LIN {X 0,Y 448.468,Z 1012.095,A -85,B 0,C 180,E1 21481.185,E2 21481.185} C_VEL
LIN {X 0,Y 450.791,Z 994.348,A -85,B 0,C 180,E1 21478.882,E2 21478.882} C_VEL
LIN {X 0,Y 453.171,Z 976.212,A -85,B 0,C 180,E1 21476.826,E2 21476.826} C_VEL
LIN {X 0,Y 455.624,Z 956.598,A -85,B 0,C 180,E1 21474.938,E2 21474.938} C_VEL
LIN {X 0,Y 458.226,Z 934.729,A -85,B 0,C 180,E1 21473.126,E2 21473.126} C_VEL
LIN {X 0,Y 460.541,Z 914.08,A -85,B 0,C 180,E1 21471.667,E2 21471.667} C_VEL
LIN {X 0,Y 462.807,Z 891.263,A -85,B 0,C 180,E1 21470.327,E2 21470.327} C_VEL
LIN {X 0,Y 464.943,Z 868.015,A -85,B 0,C 180,E1 21469.198,E2 21469.198} C_VEL
LIN {X 0,Y 466.739,Z 845.323,A -85,B 0,C 180,E1 21468.323,E2 21468.323} C_VEL
LIN {X 0,Y 468.364,Z 820.403,A -85,B 0,C 180,E1 21467.596,E2 21467.596} C_VEL
LIN {X 0,Y 469.433,Z 794.902,A -85,B 0,C 180,E1 21467.062,E2 21467.062} C_VEL
LIN {X 0,Y 475.124,Z 590.761,A -85,B 0,C 180,E1 21463.377,E2 21463.377} C_VEL
LIN {X 0,Y 477.769,Z 494.434,A -85,B 0,C 180,E1 21461.609,E2 21461.609} C_VEL
LIN {X 0,Y 474.776,Z 465.725,A -85,B 0,C 180,E1 21460.637,E2 21460.637} C_VEL
LIN {X 0,Y 475.531,Z 455.632,A -85,B 0,C 180,E1 21460.006,E2 21460.006} C_VEL
LIN {X 0,Y 466.495,Z 437.235,A -85,B 0,C 180,E1 21457.496,E2 21457.496} C_VEL
LIN {X 0,Y 457.538,Z 420.696,A -85,B 0,C 180,E1 21454.928,E2 21454.928} C_VEL
LIN {X 0,Y 449.786,Z 407.184,A -85,B 0,C 180,E1 21452.544,E2 21452.544} C_VEL
LIN {X 0,Y 447.205,Z 402.648,A -85,B 0,C 180,E1 21451.695,E2 21451.695} C_VEL
LIN {X 0,Y 444.59,Z 398.544,A -85,B 0,C 180,E1 21450.847,E2 21450.847} C_VEL
LIN {X 0,Y 443.917,Z 397.22,A -85,B 0,C 180,E1 21450.599,E2 21450.599} C_VEL
LIN {X 0,Y 441.681,Z 394.126,A -85,B 0,C 180,E1 21449.885,E2 21449.885} C_VEL
LIN {X 0,Y 441.204,Z 392.302,A -85,B 0,C 180,E1 21449.514,E2 21449.514} C_VEL
LIN {X 0,Y 441.121,Z 392.05,A -85,B 0,C 180,E1 21445.941,E2 21445.941} C_VEL
LIN {X 0,Y 441.125,Z 392.099,A -85,B 0,C 180,E1 21442.242,E2 21442.242} C_VEL
LIN {X 0,Y 441.157,Z 392.047,A -85,B 0,C 180,E1 21438.636,E2 21438.636} C_VEL
LIN {X 0,Y 441.161,Z 392.066,A -85,B 0,C 180,E1 21434.973,E2 21434.973} C_VEL
LIN {X 0,Y 441.122,Z 392.06,A -85,B 0,C 180,E1 21431.373,E2 21431.373} C_VEL
LIN {X 0,Y 441.124,Z 392.081,A -85,B 0,C 180,E1 21427.554,E2 21427.554} C_VEL
LIN {X 0,Y 441.164,Z 392.078,A -85,B 0,C 180,E1 21424.028,E2 21424.028} C_VEL
LIN {X 0,Y 441.174,Z 392.079,A -85,B 0,C 180,E1 21420.259,E2 21420.259} C_VEL
LIN {X 0,Y 441.132,Z 392.084,A -85,B 0,C 180,E1 21416.621,E2 21416.621} C_VEL
LIN {X 0,Y 441.128,Z 392.084,A -85,B 0,C 180,E1 21412.969,E2 21412.969} C_VEL
LIN {X 0,Y 441.171,Z 392.08,A -85,B 0,C 180,E1 21409.421,E2 21409.421} C_VEL
LIN {X 0,Y 441.17,Z 392.083,A -85,B 0,C 180,E1 21405.697,E2 21405.697} C_VEL
LIN {X 0,Y 441.133,Z 392.089,A -85,B 0,C 180,E1 21402.046,E2 21402.046} C_VEL
LIN {X 0,Y 441.131,Z 392.086,A -85,B 0,C 180,E1 21398.318,E2 21398.318} C_VEL
LIN {X 0,Y 441.17,Z 392.081,A -85,B 0,C 180,E1 21394.728,E2 21394.728} C_VEL
LIN {X 0,Y 441.163,Z 392.055,A -85,B 0,C 180,E1 21391.135,E2 21391.135} C_VEL
LIN {X 0,Y 441.135,Z 392.085,A -85,B 0,C 180,E1 21387.476,E2 21387.476} C_VEL
LIN {X 0,Y 441.131,Z 392.048,A -85,B 0,C 180,E1 21383.731,E2 21383.731} C_VEL
LIN {X 0,Y 441.177,Z 392.355,A -85,B 0,C 180,E1 21381.087,E2 21381.087} C_VEL
LIN {X 0,Y 442.762,Z 395.916,A -85,B 0,C 180,E1 21380.276,E2 21380.276} C_VEL
LIN {X 0,Y 443.854,Z 397.437,A -85,B 0,C 180,E1 21379.889,E2 21379.889} C_VEL
LIN {X 0,Y 445.782,Z 401.239,A -85,B 0,C 180,E1 21379.085,E2 21379.085} C_VEL
LIN {X 0,Y 446.794,Z 403.101,A -85,B 0,C 180,E1 21378.687,E2 21378.687} C_VEL
LIN {X 0,Y 451.901,Z 412.956,A -85,B 0,C 180,E1 21376.694,E2 21376.694} C_VEL
LIN {X 0,Y 457.667,Z 424.557,A -85,B 0,C 180,E1 21374.531,E2 21374.531} C_VEL
LIN {X 0,Y 464.484,Z 439.37,A -85,B 0,C 180,E1 21372.026,E2 21372.026} C_VEL
LIN {X 0,Y 468.3,Z 448.451,A -85,B 0,C 180,E1 21370.633,E2 21370.633} C_VEL
LIN {X 0,Y 466.212,Z 469.982,A -85,B 0,C 180,E1 21368.876,E2 21368.876} C_VEL
LIN {X 0,Y 471.019,Z 499.481,A -85,B 0,C 180,E1 21367.741,E2 21367.741} C_VEL
LIN {X 0,Y 468.419,Z 640.813,A -85,B 0,C 180,E1 21365.511,E2 21365.511} C_VEL
LIN {X 0,Y 467.57,Z 648.523,A -85,B 0,C 180,E1 21365.47,E2 21365.47} C_VEL
LIN {X 0,Y 462.514,Z 669.112,A -85,B 0,C 180,E1 21365.661,E2 21365.661} C_VEL
LIN {X 0,Y 461.847,Z 675.731,A -85,B 0,C 180,E1 21365.619,E2 21365.619} C_VEL
LIN {X 0,Y 460.705,Z 743.485,A -85,B 0,C 180,E1 21364.531,E2 21364.531} C_VEL
LIN {X 0,Y 459.78,Z 763.748,A -85,B 0,C 180,E1 21363.979,E2 21363.979} C_VEL
LIN {X 0,Y 458.394,Z 783.122,A -85,B 0,C 180,E1 21363.232,E2 21363.232} C_VEL
LIN {X 0,Y 456.607,Z 801.726,A -85,B 0,C 180,E1 21362.297,E2 21362.297} C_VEL
LIN {X 0,Y 454.373,Z 820.148,A -85,B 0,C 180,E1 21361.129,E2 21361.129} C_VEL
LIN {X 0,Y 451.88,Z 837.225,A -85,B 0,C 180,E1 21359.785,E2 21359.785} C_VEL
LIN {X 0,Y 449.157,Z 853.741,A -85,B 0,C 180,E1 21358.22,E2 21358.22} C_VEL
LIN {X 0,Y 446.413,Z 869.137,A -85,B 0,C 180,E1 21356.469,E2 21356.469} C_VEL
LIN {X 0,Y 443.615,Z 883.656,A -85,B 0,C 180,E1 21354.502,E2 21354.502} C_VEL
LIN {X 0,Y 440.907,Z 897.352,A -85,B 0,C 180,E1 21352.254,E2 21352.254} C_VEL
LIN {X 0,Y 438.611,Z 908.804,A -85,B 0,C 180,E1 21349.995,E2 21349.995} C_VEL
LIN {X 0,Y 436.583,Z 919.459,A -85,B 0,C 180,E1 21347.459,E2 21347.459} C_VEL
LIN {X 0,Y 434.978,Z 928.589,A -85,B 0,C 180,E1 21344.783,E2 21344.783} C_VEL
LIN {X 0,Y 433.854,Z 935.893,A -85,B 0,C 180,E1 21342.106,E2 21342.106} C_VEL
LIN {X 0,Y 433.096,Z 942.058,A -85,B 0,C 180,E1 21339.166,E2 21339.166} C_VEL
LIN {X 0,Y 432.688,Z 946.439,A -85,B 0,C 180,E1 21336.235,E2 21336.235} C_VEL
LIN {X 0,Y 432.469,Z 949.098,A -85,B 0,C 180,E1 21333.314,E2 21333.314} C_VEL
LIN {X 0,Y 432.408,Z 950.106,A -85,B 0,C 180,E1 21330.53,E2 21330.53} C_VEL
LIN {X 0,Y 432.438,Z 949.614,A -85,B 0,C 180,E1 21327.615,E2 21327.615} C_VEL
LIN {X 0,Y 432.577,Z 947.513,A -85,B 0,C 180,E1 21324.695,E2 21324.695} C_VEL
LIN {X 0,Y 432.899,Z 943.973,A -85,B 0,C 180,E1 21321.901,E2 21321.901} C_VEL
LIN {X 0,Y 433.461,Z 938.858,A -85,B 0,C 180,E1 21319.097,E2 21319.097} C_VEL
LIN {X 0,Y 434.522,Z 931.627,A -85,B 0,C 180,E1 21316.154,E2 21316.154} C_VEL
LIN {X 0,Y 435.898,Z 923.218,A -85,B 0,C 180,E1 21313.475,E2 21313.475} C_VEL
LIN {X 0,Y 437.744,Z 913.352,A -85,B 0,C 180,E1 21310.936,E2 21310.936} C_VEL
LIN {X 0,Y 439.944,Z 902.052,A -85,B 0,C 180,E1 21308.537,E2 21308.537} C_VEL
LIN {X 0,Y 442.345,Z 890.111,A -85,B 0,C 180,E1 21306.416,E2 21306.416} C_VEL
LIN {X 0,Y 445.131,Z 875.915,A -85,B 0,C 180,E1 21304.309,E2 21304.309} C_VEL
LIN {X 0,Y 448.018,Z 860.412,A -85,B 0,C 180,E1 21302.406,E2 21302.406} C_VEL
LIN {X 0,Y 450.706,Z 844.615,A -85,B 0,C 180,E1 21300.787,E2 21300.787} C_VEL
LIN {X 0,Y 453.397,Z 827.134,A -85,B 0,C 180,E1 21299.301,E2 21299.301} C_VEL
LIN {X 0,Y 455.721,Z 809.616,A -85,B 0,C 180,E1 21298.078,E2 21298.078} C_VEL
LIN {X 0,Y 457.698,Z 791.119,A -85,B 0,C 180,E1 21297.047,E2 21297.047} C_VEL
LIN {X 0,Y 459.274,Z 772.031,A -85,B 0,C 180,E1 21296.223,E2 21296.223} C_VEL
LIN {X 0,Y 460.396,Z 751.626,A -85,B 0,C 180,E1 21295.574,E2 21295.574} C_VEL
LIN {X 0,Y 460.968,Z 731.073,A -85,B 0,C 180,E1 21295.147,E2 21295.147} C_VEL
LIN {X 0,Y 465.125,Z 504.024,A -85,B 0,C 180,E1 21291.563,E2 21291.563} C_VEL
LIN {X 0,Y 465.006,Z 498.899,A -85,B 0,C 180,E1 21291.45,E2 21291.45} C_VEL
LIN {X 0,Y 460.181,Z 468.723,A -85,B 0,C 180,E1 21290.217,E2 21290.217} C_VEL
LIN {X 0,Y 461.91,Z 451.947,A -85,B 0,C 180,E1 21288.792,E2 21288.792} C_VEL
LIN {X 0,Y 454.83,Z 435.65,A -85,B 0,C 180,E1 21286.141,E2 21286.141} C_VEL
LIN {X 0,Y 447.451,Z 420.273,A -85,B 0,C 180,E1 21283.316,E2 21283.316} C_VEL
LIN {X 0,Y 440.681,Z 407.247,A -85,B 0,C 180,E1 21280.63,E2 21280.63} C_VEL
LIN {X 0,Y 437.714,Z 401.938,A -85,B 0,C 180,E1 21279.423,E2 21279.423} C_VEL
LIN {X 0,Y 435.539,Z 397.815,A -85,B 0,C 180,E1 21278.472,E2 21278.472} C_VEL
LIN {X 0,Y 433.601,Z 394.615,A -85,B 0,C 180,E1 21277.668,E2 21277.668} C_VEL
LIN {X 0,Y 433.24,Z 393.102,A -85,B 0,C 180,E1 21277.234,E2 21277.234} C_VEL
LIN {X 0,Y 433.25,Z 393.077,A -85,B 0,C 180,E1 21273.475,E2 21273.475} C_VEL
LIN {X 0,Y 433.203,Z 393.029,A -85,B 0,C 180,E1 21269.751,E2 21269.751} C_VEL
LIN {X 0,Y 433.199,Z 393.076,A -85,B 0,C 180,E1 21266.011,E2 21266.011} C_VEL
LIN {X 0,Y 433.206,Z 393.071,A -85,B 0,C 180,E1 21262.242,E2 21262.242} C_VEL
LIN {X 0,Y 433.243,Z 393.068,A -85,B 0,C 180,E1 21258.572,E2 21258.572} C_VEL
LIN {X 0,Y 433.227,Z 393.068,A -85,B 0,C 180,E1 21254.844,E2 21254.844} C_VEL
LIN {X 0,Y 433.195,Z 393.07,A -85,B 0,C 180,E1 21251.18,E2 21251.18} C_VEL
LIN {X 0,Y 433.193,Z 393.071,A -85,B 0,C 180,E1 21247.427,E2 21247.427} C_VEL
LIN {X 0,Y 433.23,Z 393.068,A -85,B 0,C 180,E1 21243.838,E2 21243.838} C_VEL
LIN {X 0,Y 433.248,Z 393.067,A -85,B 0,C 180,E1 21240,E2 21240} C_VEL
LIN {X 0,Y 433.203,Z 393.073,A -85,B 0,C 180,E1 21236.295,E2 21236.295} C_VEL
LIN {X 0,Y 433.187,Z 393.073,A -85,B 0,C 180,E1 21232.574,E2 21232.574} C_VEL
LIN {X 0,Y 433.195,Z 393.053,A -85,B 0,C 180,E1 21228.821,E2 21228.821} C_VEL
LIN {X 0,Y 433.239,Z 393.044,A -85,B 0,C 180,E1 21225.157,E2 21225.157} C_VEL
LIN {X 0,Y 433.213,Z 393.034,A -85,B 0,C 180,E1 21221.428,E2 21221.428} C_VEL
LIN {X 0,Y 433.188,Z 393.084,A -85,B 0,C 180,E1 21217.755,E2 21217.755} C_VEL
LIN {X 0,Y 433.18,Z 393.037,A -85,B 0,C 180,E1 21213.882,E2 21213.882} C_VEL
LIN {X 0,Y 433.206,Z 393.185,A -85,B 0,C 180,E1 21212.061,E2 21212.061} C_VEL
LIN {X 0,Y 433.375,Z 394.077,A -85,B 0,C 180,E1 21211.774,E2 21211.774} C_VEL
LIN {X 0,Y 434.939,Z 397.128,A -85,B 0,C 180,E1 21211.135,E2 21211.135} C_VEL
LIN {X 0,Y 436.493,Z 398.918,A -85,B 0,C 180,E1 21210.647,E2 21210.647} C_VEL
LIN {X 0,Y 438.48,Z 402.68,A -85,B 0,C 180,E1 21209.891,E2 21209.891} C_VEL
LIN {X 0,Y 439.64,Z 404.191,A -85,B 0,C 180,E1 21209.526,E2 21209.526} C_VEL
LIN {X 0,Y 448.134,Z 418.764,A -85,B 0,C 180,E1 21206.711,E2 21206.711} C_VEL
LIN {X 0,Y 457.182,Z 435.066,A -85,B 0,C 180,E1 21203.964,E2 21203.964} C_VEL
LIN {X 0,Y 466.517,Z 453.526,A -85,B 0,C 180,E1 21201.258,E2 21201.258} C_VEL
LIN {X 0,Y 469.372,Z 459.759,A -85,B 0,C 180,E1 21200.437,E2 21200.437} C_VEL
LIN {X 0,Y 468.908,Z 467.207,A -85,B 0,C 180,E1 21200.003,E2 21200.003} C_VEL
LIN {X 0,Y 471.972,Z 498.397,A -85,B 0,C 180,E1 21198.963,E2 21198.963} C_VEL
LIN {X 0,Y 465.873,Z 694.074,A -85,B 0,C 180,E1 21195.358,E2 21195.358} C_VEL
LIN {X 0,Y 462.333,Z 810.411,A -85,B 0,C 180,E1 21193.203,E2 21193.203} C_VEL
LIN {X 0,Y 460.677,Z 834.598,A -85,B 0,C 180,E1 21192.553,E2 21192.553} C_VEL
LIN {X 0,Y 458.633,Z 859.758,A -85,B 0,C 180,E1 21191.63,E2 21191.63} C_VEL
LIN {X 0,Y 456.391,Z 883.845,A -85,B 0,C 180,E1 21190.518,E2 21190.518} C_VEL
LIN {X 0,Y 454.058,Z 905.996,A -85,B 0,C 180,E1 21189.258,E2 21189.258} C_VEL
LIN {X 0,Y 451.451,Z 929.158,A -85,B 0,C 180,E1 21187.682,E2 21187.682} C_VEL
LIN {X 0,Y 448.984,Z 949.425,A -85,B 0,C 180,E1 21186.063,E2 21186.063} C_VEL
LIN {X 0,Y 446.433,Z 969.107,A -85,B 0,C 180,E1 21184.205,E2 21184.205} C_VEL
LIN {X 0,Y 443.953,Z 987.875,A -85,B 0,C 180,E1 21182.177,E2 21182.177} C_VEL
LIN {X 0,Y 441.759,Z 1003.879,A -85,B 0,C 180,E1 21180.164,E2 21180.164} C_VEL
LIN {X 0,Y 439.529,Z 1020.382,A -85,B 0,C 180,E1 21177.797,E2 21177.797} C_VEL
LIN {X 0,Y 437.627,Z 1034.57,A -85,B 0,C 180,E1 21175.438,E2 21175.438} C_VEL
LIN {X 0,Y 436.501,Z 1043.063,A -85,B 0,C 180,E1 21173.775,E2 21173.775} C_VEL
LIN {X 0,Y 434.82,Z 1055.286,A -85,B 0,C 180,E1 21170.881,E2 21170.881} C_VEL
LIN {X 0,Y 433.661,Z 1065.058,A -85,B 0,C 180,E1 21168.135,E2 21168.135} C_VEL
LIN {X 0,Y 432.778,Z 1074.344,A -85,B 0,C 180,E1 21164.996,E2 21164.996} C_VEL
LIN {X 0,Y 432.319,Z 1080.863,A -85,B 0,C 180,E1 21162.285,E2 21162.285} C_VEL
LIN {X 0,Y 432.046,Z 1086.635,A -85,B 0,C 180,E1 21159.189,E2 21159.189} C_VEL
LIN {X 0,Y 431.946,Z 1090.278,A -85,B 0,C 180,E1 21156.513,E2 21156.513} C_VEL
LIN {X 0,Y 431.89,Z 1092.916,A -85,B 0,C 180,E1 21153.451,E2 21153.451} C_VEL
LIN {X 0,Y 431.89,Z 1093.849,A -85,B 0,C 180,E1 21150.929,E2 21150.929} C_VEL
LIN {X 0,Y 431.906,Z 1093.69,A -85,B 0,C 180,E1 21148.143,E2 21148.143} C_VEL
LIN {X 0,Y 431.911,Z 1091.954,A -85,B 0,C 180,E1 21145.219,E2 21145.219} C_VEL
LIN {X 0,Y 431.947,Z 1089.16,A -85,B 0,C 180,E1 21142.552,E2 21142.552} C_VEL
LIN {X 0,Y 432.131,Z 1084.335,A -85,B 0,C 180,E1 21139.468,E2 21139.468} C_VEL
LIN {X 0,Y 432.457,Z 1078.689,A -85,B 0,C 180,E1 21136.745,E2 21136.745} C_VEL
LIN {X 0,Y 433.109,Z 1070.549,A -85,B 0,C 180,E1 21133.641,E2 21133.641} C_VEL
LIN {X 0,Y 434.063,Z 1061.522,A -85,B 0,C 180,E1 21130.808,E2 21130.808} C_VEL
LIN {X 0,Y 435.397,Z 1050.859,A -85,B 0,C 180,E1 21128.018,E2 21128.018} C_VEL
LIN {X 0,Y 436.867,Z 1040.444,A -85,B 0,C 180,E1 21125.671,E2 21125.671} C_VEL
LIN {X 0,Y 438.484,Z 1028.182,A -85,B 0,C 180,E1 21123.453,E2 21123.453} C_VEL
LIN {X 0,Y 440.51,Z 1012.885,A -85,B 0,C 180,E1 21121.088,E2 21121.088} C_VEL
LIN {X 0,Y 442.927,Z 995.3,A -85,B 0,C 180,E1 21118.721,E2 21118.721} C_VEL
LIN {X 0,Y 445.296,Z 977.664,A -85,B 0,C 180,E1 21116.681,E2 21116.681} C_VEL
LIN {X 0,Y 447.942,Z 957.612,A -85,B 0,C 180,E1 21114.681,E2 21114.681} C_VEL
LIN {X 0,Y 450.477,Z 937.455,A -85,B 0,C 180,E1 21112.943,E2 21112.943} C_VEL
LIN {X 0,Y 452.963,Z 916.014,A -85,B 0,C 180,E1 21111.389,E2 21111.389} C_VEL
LIN {X 0,Y 455.519,Z 892.134,A -85,B 0,C 180,E1 21109.929,E2 21109.929} C_VEL
LIN {X 0,Y 457.861,Z 868.453,A -85,B 0,C 180,E1 21108.738,E2 21108.738} C_VEL
LIN {X 0,Y 459.897,Z 845.034,A -85,B 0,C 180,E1 21107.8,E2 21107.8} C_VEL
LIN {X 0,Y 461.703,Z 820.565,A -85,B 0,C 180,E1 21107.048,E2 21107.048} C_VEL
LIN {X 0,Y 462.89,Z 796.443,A -85,B 0,C 180,E1 21106.513,E2 21106.513} C_VEL
LIN {X 0,Y 469.226,Z 586.155,A -85,B 0,C 180,E1 21102.65,E2 21102.65} C_VEL
LIN {X 0,Y 471.857,Z 495.824,A -85,B 0,C 180,E1 21100.973,E2 21100.973} C_VEL
LIN {X 0,Y 468.83,Z 465.707,A -85,B 0,C 180,E1 21099.935,E2 21099.935} C_VEL
LIN {X 0,Y 469.264,Z 459.399,A -85,B 0,C 180,E1 21099.528,E2 21099.528} C_VEL
LIN {X 0,Y 460.765,Z 442.036,A -85,B 0,C 180,E1 21097.103,E2 21097.103} C_VEL
LIN {X 0,Y 451.956,Z 425.626,A -85,B 0,C 180,E1 21094.495,E2 21094.495} C_VEL
LIN {X 0,Y 444.665,Z 412.9,A -85,B 0,C 180,E1 21092.202,E2 21092.202} C_VEL
LIN {X 0,Y 441.33,Z 407.353,A -85,B 0,C 180,E1 21091.1,E2 21091.1} C_VEL
LIN {X 0,Y 439.258,Z 403.53,A -85,B 0,C 180,E1 21090.352,E2 21090.352} C_VEL
LIN {X 0,Y 437.001,Z 400.277,A -85,B 0,C 180,E1 21089.605,E2 21089.605} C_VEL
LIN {X 0,Y 436.11,Z 398.272,A -85,B 0,C 180,E1 21089.231,E2 21089.231} C_VEL
LIN {X 0,Y 433.852,Z 395.425,A -85,B 0,C 180,E1 21088.493,E2 21088.493} C_VEL
LIN {X 0,Y 433.221,Z 393.312,A -85,B 0,C 180,E1 21088.049,E2 21088.049} C_VEL
LIN {X 0,Y 433.199,Z 393.038,A -85,B 0,C 180,E1 21084.693,E2 21084.693} C_VEL
LIN {X 0,Y 433.235,Z 393.042,A -85,B 0,C 180,E1 21081.102,E2 21081.102} C_VEL
LIN {X 0,Y 433.202,Z 393.07,A -85,B 0,C 180,E1 21077.321,E2 21077.321} C_VEL
LIN {X 0,Y 433.178,Z 393.028,A -85,B 0,C 180,E1 21073.649,E2 21073.649} C_VEL
LIN {X 0,Y 433.2,Z 393.081,A -85,B 0,C 180,E1 21069.968,E2 21069.968} C_VEL
LIN {X 0,Y 433.247,Z 393.074,A -85,B 0,C 180,E1 21066.36,E2 21066.36} C_VEL
LIN {X 0,Y 433.219,Z 393.081,A -85,B 0,C 180,E1 21062.513,E2 21062.513} C_VEL
LIN {X 0,Y 433.188,Z 393.085,A -85,B 0,C 180,E1 21058.942,E2 21058.942} C_VEL
LIN {X 0,Y 433.192,Z 393.086,A -85,B 0,C 180,E1 21055.101,E2 21055.101} C_VEL
LIN {X 0,Y 433.233,Z 393.076,A -85,B 0,C 180,E1 21051.506,E2 21051.506} C_VEL
LIN {X 0,Y 433.233,Z 393.074,A -85,B 0,C 180,E1 21047.741,E2 21047.741} C_VEL
LIN {X 0,Y 433.192,Z 393.079,A -85,B 0,C 180,E1 21044.195,E2 21044.195} C_VEL
LIN {X 0,Y 433.192,Z 393.083,A -85,B 0,C 180,E1 21040.343,E2 21040.343} C_VEL
LIN {X 0,Y 433.222,Z 393.081,A -85,B 0,C 180,E1 21036.719,E2 21036.719} C_VEL
LIN {X 0,Y 433.25,Z 393.083,A -85,B 0,C 180,E1 21032.958,E2 21032.958} C_VEL
LIN {X 0,Y 433.198,Z 393.03,A -85,B 0,C 180,E1 21029.33,E2 21029.33} C_VEL
LIN {X 0,Y 433.193,Z 393.059,A -85,B 0,C 180,E1 21025.722,E2 21025.722} C_VEL
LIN {X 0,Y 433.275,Z 393.272,A -85,B 0,C 180,E1 21022.547,E2 21022.547} C_VEL
LIN {X 0,Y 434.562,Z 396.641,A -85,B 0,C 180,E1 21021.762,E2 21021.762} C_VEL
LIN {X 0,Y 436.025,Z 398.504,A -85,B 0,C 180,E1 21021.23,E2 21021.23} C_VEL
LIN {X 0,Y 437.837,Z 402.121,A -85,B 0,C 180,E1 21020.421,E2 21020.421} C_VEL
LIN {X 0,Y 439.101,Z 404.577,A -85,B 0,C 180,E1 21019.878,E2 21019.878} C_VEL
LIN {X 0,Y 441.467,Z 408.736,A -85,B 0,C 180,E1 21018.943,E2 21018.943} C_VEL
LIN {X 0,Y 447.932,Z 421.252,A -85,B 0,C 180,E1 21016.39,E2 21016.39} C_VEL
LIN {X 0,Y 455.311,Z 436.855,A -85,B 0,C 180,E1 21013.558,E2 21013.558} C_VEL
LIN {X 0,Y 461.991,Z 452.277,A -85,B 0,C 180,E1 21011.069,E2 21011.069} C_VEL
LIN {X 0,Y 460.191,Z 469.857,A -85,B 0,C 180,E1 21009.622,E2 21009.622} C_VEL
LIN {X 0,Y 465.187,Z 501.003,A -85,B 0,C 180,E1 21008.394,E2 21008.394} C_VEL
LIN {X 0,Y 461.847,Z 675.731,A -85,B 0,C 180,E1 21005.619,E2 21005.619} C_VEL
LIN {X 0,Y 460.984,Z 683.439,A -85,B 0,C 180,E1 21005.58,E2 21005.58} C_VEL
LIN {X 0,Y 455.916,Z 704.017,A -85,B 0,C 180,E1 21005.776,E2 21005.776} C_VEL
LIN {X 0,Y 455.217,Z 710.635,A -85,B 0,C 180,E1 21005.736,E2 21005.736} C_VEL
LIN {X 0,Y 454.534,Z 745.79,A -85,B 0,C 180,E1 21005.136,E2 21005.136} C_VEL
LIN {X 0,Y 453.54,Z 766.188,A -85,B 0,C 180,E1 21004.56,E2 21004.56} C_VEL
LIN {X 0,Y 452.058,Z 785.284,A -85,B 0,C 180,E1 21003.798,E2 21003.798} C_VEL
LIN {X 0,Y 450.103,Z 804.155,A -85,B 0,C 180,E1 21002.822,E2 21002.822} C_VEL
LIN {X 0,Y 447.8,Z 822.219,A -85,B 0,C 180,E1 21001.649,E2 21001.649} C_VEL
LIN {X 0,Y 445.18,Z 839.286,A -85,B 0,C 180,E1 21000.28,E2 21000.28} C_VEL
LIN {X 0,Y 442.37,Z 855.414,A -85,B 0,C 180,E1 20998.72,E2 20998.72} C_VEL
LIN {X 0,Y 439.448,Z 870.944,A -85,B 0,C 180,E1 20996.922,E2 20996.922} C_VEL
LIN {X 0,Y 436.702,Z 884.518,A -85,B 0,C 180,E1 20995.06,E2 20995.06} C_VEL
LIN {X 0,Y 433.977,Z 897.535,A -85,B 0,C 180,E1 20992.915,E2 20992.915} C_VEL
LIN {X 0,Y 431.439,Z 909.484,A -85,B 0,C 180,E1 20990.565,E2 20990.565} C_VEL
LIN {X 0,Y 429.187,Z 920.585,A -85,B 0,C 180,E1 20987.91,E2 20987.91} C_VEL
LIN {X 0,Y 427.435,Z 929.8,A -85,B 0,C 180,E1 20985.188,E2 20985.188} C_VEL
LIN {X 0,Y 426.209,Z 937.166,A -85,B 0,C 180,E1 20982.464,E2 20982.464} C_VEL
LIN {X 0,Y 425.364,Z 943.114,A -85,B 0,C 180,E1 20979.607,E2 20979.607} C_VEL
LIN {X 0,Y 424.878,Z 947.533,A -85,B 0,C 180,E1 20976.622,E2 20976.622} C_VEL
LIN {X 0,Y 424.62,Z 950.195,A -85,B 0,C 180,E1 20973.78,E2 20973.78} C_VEL
LIN {X 0,Y 424.534,Z 951.432,A -85,B 0,C 180,E1 20970.81,E2 20970.81} C_VEL
LIN {X 0,Y 424.558,Z 951.106,A -85,B 0,C 180,E1 20967.841,E2 20967.841} C_VEL
LIN {X 0,Y 424.706,Z 949.346,A -85,B 0,C 180,E1 20965.003,E2 20965.003} C_VEL
LIN {X 0,Y 425.049,Z 945.883,A -85,B 0,C 180,E1 20962.022,E2 20962.022} C_VEL
LIN {X 0,Y 425.668,Z 940.742,A -85,B 0,C 180,E1 20959.068,E2 20959.068} C_VEL
LIN {X 0,Y 426.675,Z 934.284,A -85,B 0,C 180,E1 20956.309,E2 20956.309} C_VEL
LIN {X 0,Y 428.088,Z 926.192,A -85,B 0,C 180,E1 20953.584,E2 20953.584} C_VEL
LIN {X 0,Y 429.983,Z 916.692,A -85,B 0,C 180,E1 20951.001,E2 20951.001} C_VEL
LIN {X 0,Y 432.235,Z 905.82,A -85,B 0,C 180,E1 20948.562,E2 20948.562} C_VEL
LIN {X 0,Y 434.946,Z 892.994,A -85,B 0,C 180,E1 20946.196,E2 20946.196} C_VEL
LIN {X 0,Y 437.714,Z 879.534,A -85,B 0,C 180,E1 20944.132,E2 20944.132} C_VEL
LIN {X 0,Y 440.615,Z 864.947,A -85,B 0,C 180,E1 20942.252,E2 20942.252} C_VEL
LIN {X 0,Y 443.487,Z 849.341,A -85,B 0,C 180,E1 20940.561,E2 20940.561} C_VEL
LIN {X 0,Y 446.277,Z 832.59,A -85,B 0,C 180,E1 20939.057,E2 20939.057} C_VEL
LIN {X 0,Y 448.798,Z 814.844,A -85,B 0,C 180,E1 20937.753,E2 20937.753} C_VEL
LIN {X 0,Y 450.993,Z 796.221,A -85,B 0,C 180,E1 20936.645,E2 20936.645} C_VEL
LIN {X 0,Y 452.798,Z 776.87,A -85,B 0,C 180,E1 20935.745,E2 20935.745} C_VEL
LIN {X 0,Y 454.099,Z 757.056,A -85,B 0,C 180,E1 20935.062,E2 20935.062} C_VEL
LIN {X 0,Y 454.763,Z 736.951,A -85,B 0,C 180,E1 20934.596,E2 20934.596} C_VEL
LIN {X 0,Y 459.428,Z 501.652,A -85,B 0,C 180,E1 20930.825,E2 20930.825} C_VEL
LIN {X 0,Y 454.252,Z 468.861,A -85,B 0,C 180,E1 20929.467,E2 20929.467} C_VEL
LIN {X 0,Y 455.628,Z 455.879,A -85,B 0,C 180,E1 20928.35,E2 20928.35} C_VEL
LIN {X 0,Y 448.298,Z 438.984,A -85,B 0,C 180,E1 20925.538,E2 20925.538} C_VEL
LIN {X 0,Y 441.704,Z 425.283,A -85,B 0,C 180,E1 20922.95,E2 20922.95} C_VEL
LIN {X 0,Y 435.753,Z 413.46,A -85,B 0,C 180,E1 20920.494,E2 20920.494} C_VEL
LIN {X 0,Y 432.121,Z 407.113,A -85,B 0,C 180,E1 20919.004,E2 20919.004} C_VEL
LIN {X 0,Y 430.277,Z 403.623,A -85,B 0,C 180,E1 20918.179,E2 20918.179} C_VEL
LIN {X 0,Y 428.446,Z 400.267,A -85,B 0,C 180,E1 20917.356,E2 20917.356} C_VEL
LIN {X 0,Y 427.9,Z 399.033,A -85,B 0,C 180,E1 20917.075,E2 20917.075} C_VEL
LIN {X 0,Y 425.896,Z 396.306,A -85,B 0,C 180,E1 20916.272,E2 20916.272} C_VEL
LIN {X 0,Y 425.331,Z 394.346,A -85,B 0,C 180,E1 20915.804,E2 20915.804} C_VEL
LIN {X 0,Y 425.258,Z 394.04,A -85,B 0,C 180,E1 20914.353,E2 20914.353} C_VEL
LIN {X 0,Y 425.265,Z 394.016,A -85,B 0,C 180,E1 20910.624,E2 20910.624} C_VEL
LIN {X 0,Y 425.311,Z 394.072,A -85,B 0,C 180,E1 20906.983,E2 20906.983} C_VEL
LIN {X 0,Y 425.302,Z 394.065,A -85,B 0,C 180,E1 20903.117,E2 20903.117} C_VEL
LIN {X 0,Y 425.269,Z 394.066,A -85,B 0,C 180,E1 20899.361,E2 20899.361} C_VEL
LIN {X 0,Y 425.257,Z 394.066,A -85,B 0,C 180,E1 20895.688,E2 20895.688} C_VEL
LIN {X 0,Y 425.281,Z 394.061,A -85,B 0,C 180,E1 20892.028,E2 20892.028} C_VEL
LIN {X 0,Y 425.313,Z 394.058,A -85,B 0,C 180,E1 20888.219,E2 20888.219} C_VEL
LIN {X 0,Y 425.28,Z 394.064,A -85,B 0,C 180,E1 20884.45,E2 20884.45} C_VEL
LIN {X 0,Y 425.253,Z 394.071,A -85,B 0,C 180,E1 20880.809,E2 20880.809} C_VEL
LIN {X 0,Y 425.252,Z 394.069,A -85,B 0,C 180,E1 20876.9,E2 20876.9} C_VEL
LIN {X 0,Y 425.279,Z 394.065,A -85,B 0,C 180,E1 20873.25,E2 20873.25} C_VEL
LIN {X 0,Y 425.297,Z 394.058,A -85,B 0,C 180,E1 20869.571,E2 20869.571} C_VEL
LIN {X 0,Y 425.257,Z 394.019,A -85,B 0,C 180,E1 20865.847,E2 20865.847} C_VEL
LIN {X 0,Y 425.246,Z 394.041,A -85,B 0,C 180,E1 20862.202,E2 20862.202} C_VEL
LIN {X 0,Y 425.263,Z 394.042,A -85,B 0,C 180,E1 20858.483,E2 20858.483} C_VEL
LIN {X 0,Y 425.294,Z 394.015,A -85,B 0,C 180,E1 20854.816,E2 20854.816} C_VEL
LIN {X 0,Y 425.294,Z 394.362,A -85,B 0,C 180,E1 20853.545,E2 20853.545} C_VEL
LIN {X 0,Y 426.96,Z 398.008,A -85,B 0,C 180,E1 20852.678,E2 20852.678} C_VEL
LIN {X 0,Y 428.482,Z 399.64,A -85,B 0,C 180,E1 20852.178,E2 20852.178} C_VEL
LIN {X 0,Y 430.326,Z 403.372,A -85,B 0,C 180,E1 20851.404,E2 20851.404} C_VEL
LIN {X 0,Y 431.832,Z 405.265,A -85,B 0,C 180,E1 20850.907,E2 20850.907} C_VEL
LIN {X 0,Y 434.233,Z 409.398,A -85,B 0,C 180,E1 20850.023,E2 20850.023} C_VEL
LIN {X 0,Y 438.552,Z 416.859,A -85,B 0,C 180,E1 20848.506,E2 20848.506} C_VEL
LIN {X 0,Y 443.384,Z 425.066,A -85,B 0,C 180,E1 20846.926,E2 20846.926} C_VEL
LIN {X 0,Y 451.941,Z 440.635,A -85,B 0,C 180,E1 20844.264,E2 20844.264} C_VEL
LIN {X 0,Y 461.147,Z 459.091,A -85,B 0,C 180,E1 20841.518,E2 20841.518} C_VEL
LIN {X 0,Y 463.174,Z 463.478,A -85,B 0,C 180,E1 20840.925,E2 20840.925} C_VEL
LIN {X 0,Y 463.074,Z 467.74,A -85,B 0,C 180,E1 20840.701,E2 20840.701} C_VEL
LIN {X 0,Y 466.123,Z 499.761,A -85,B 0,C 180,E1 20839.614,E2 20839.614} C_VEL
LIN {X 0,Y 459.725,Z 693.452,A -85,B 0,C 180,E1 20836.004,E2 20836.004} C_VEL
LIN {X 0,Y 455.951,Z 809.256,A -85,B 0,C 180,E1 20833.823,E2 20833.823} C_VEL
LIN {X 0,Y 454.215,Z 833.206,A -85,B 0,C 180,E1 20833.172,E2 20833.172} C_VEL
LIN {X 0,Y 452.033,Z 857.97,A -85,B 0,C 180,E1 20832.255,E2 20832.255} C_VEL
LIN {X 0,Y 449.685,Z 881.129,A -85,B 0,C 180,E1 20831.159,E2 20831.159} C_VEL
LIN {X 0,Y 446.945,Z 904.721,A -85,B 0,C 180,E1 20829.778,E2 20829.778} C_VEL
LIN {X 0,Y 444.165,Z 928.038,A -85,B 0,C 180,E1 20828.165,E2 20828.165} C_VEL
LIN {X 0,Y 441.538,Z 948.91,A -85,B 0,C 180,E1 20826.472,E2 20826.472} C_VEL
LIN {X 0,Y 438.845,Z 968.868,A -85,B 0,C 180,E1 20824.564,E2 20824.564} C_VEL
LIN {X 0,Y 436.154,Z 988.289,A -85,B 0,C 180,E1 20822.402,E2 20822.402} C_VEL
LIN {X 0,Y 433.859,Z 1004.571,A -85,B 0,C 180,E1 20820.312,E2 20820.312} C_VEL
LIN {X 0,Y 431.575,Z 1020.849,A -85,B 0,C 180,E1 20817.904,E2 20817.904} C_VEL
LIN {X 0,Y 429.738,Z 1034.112,A -85,B 0,C 180,E1 20815.643,E2 20815.643} C_VEL
LIN {X 0,Y 427.873,Z 1048.414,A -85,B 0,C 180,E1 20812.825,E2 20812.825} C_VEL
LIN {X 0,Y 426.929,Z 1056.269,A -85,B 0,C 180,E1 20810.997,E2 20810.997} C_VEL
LIN {X 0,Y 425.815,Z 1065.172,A -85,B 0,C 180,E1 20808.446,E2 20808.446} C_VEL
LIN {X 0,Y 424.868,Z 1074.344,A -85,B 0,C 180,E1 20805.282,E2 20805.282} C_VEL
LIN {X 0,Y 424.342,Z 1081.165,A -85,B 0,C 180,E1 20802.382,E2 20802.382} C_VEL
LIN {X 0,Y 424.051,Z 1086.842,A -85,B 0,C 180,E1 20799.226,E2 20799.226} C_VEL
LIN {X 0,Y 423.947,Z 1090.438,A -85,B 0,C 180,E1 20796.5,E2 20796.5} C_VEL
LIN {X 0,Y 423.888,Z 1092.984,A -85,B 0,C 180,E1 20793.381,E2 20793.381} C_VEL
LIN {X 0,Y 423.887,Z 1093.871,A -85,B 0,C 180,E1 20790.811,E2 20790.811} C_VEL
LIN {X 0,Y 423.911,Z 1093.595,A -85,B 0,C 180,E1 20787.837,E2 20787.837} C_VEL
LIN {X 0,Y 423.916,Z 1091.84,A -85,B 0,C 180,E1 20784.993,E2 20784.993} C_VEL
LIN {X 0,Y 424,Z 1088.68,A -85,B 0,C 180,E1 20782.002,E2 20782.002} C_VEL
LIN {X 0,Y 424.186,Z 1083.827,A -85,B 0,C 180,E1 20778.993,E2 20778.993} C_VEL
LIN {X 0,Y 424.596,Z 1077.516,A -85,B 0,C 180,E1 20775.963,E2 20775.963} C_VEL
LIN {X 0,Y 425.294,Z 1069.739,A -85,B 0,C 180,E1 20773.051,E2 20773.051} C_VEL
LIN {X 0,Y 426.397,Z 1060.361,A -85,B 0,C 180,E1 20770.101,E2 20770.101} C_VEL
LIN {X 0,Y 427.525,Z 1051.454,A -85,B 0,C 180,E1 20767.838,E2 20767.838} C_VEL
LIN {X 0,Y 429.066,Z 1039.395,A -85,B 0,C 180,E1 20765.342,E2 20765.342} C_VEL
LIN {X 0,Y 431.086,Z 1024.338,A -85,B 0,C 180,E1 20762.662,E2 20762.662} C_VEL
LIN {X 0,Y 433.149,Z 1009.659,A -85,B 0,C 180,E1 20760.397,E2 20760.397} C_VEL
LIN {X 0,Y 435.611,Z 992.06,A -85,B 0,C 180,E1 20758.057,E2 20758.057} C_VEL
LIN {X 0,Y 438.303,Z 973.032,A -85,B 0,C 180,E1 20755.862,E2 20755.862} C_VEL
LIN {X 0,Y 440.886,Z 953.515,A -85,B 0,C 180,E1 20753.949,E2 20753.949} C_VEL
LIN {X 0,Y 443.834,Z 930.829,A -85,B 0,C 180,E1 20752.047,E2 20752.047} C_VEL
LIN {X 0,Y 446.462,Z 909.225,A -85,B 0,C 180,E1 20750.504,E2 20750.504} C_VEL
LIN {X 0,Y 449.235,Z 884.86,A -85,B 0,C 180,E1 20749.045,E2 20749.045} C_VEL
LIN {X 0,Y 451.663,Z 861.89,A -85,B 0,C 180,E1 20747.917,E2 20747.917} C_VEL
LIN {X 0,Y 453.814,Z 838.655,A -85,B 0,C 180,E1 20747,E2 20747} C_VEL
LIN {X 0,Y 455.578,Z 814.799,A -85,B 0,C 180,E1 20746.313,E2 20746.313} C_VEL
LIN {X 0,Y 456.917,Z 782.679,A -85,B 0,C 180,E1 20745.655,E2 20745.655} C_VEL
LIN {X 0,Y 463.693,Z 572.943,A -85,B 0,C 180,E1 20741.742,E2 20741.742} C_VEL
LIN {X 0,Y 466.009,Z 497.247,A -85,B 0,C 180,E1 20740.322,E2 20740.322} C_VEL
LIN {X 0,Y 462.953,Z 465.703,A -85,B 0,C 180,E1 20739.217,E2 20739.217} C_VEL
LIN {X 0,Y 463.157,Z 463.462,A -85,B 0,C 180,E1 20739.077,E2 20739.077} C_VEL
LIN {X 0,Y 454.273,Z 445.197,A -85,B 0,C 180,E1 20736.46,E2 20736.46} C_VEL
LIN {X 0,Y 445.272,Z 428.357,A -85,B 0,C 180,E1 20733.685,E2 20733.685} C_VEL
LIN {X 0,Y 439.185,Z 417.977,A -85,B 0,C 180,E1 20731.728,E2 20731.728} C_VEL
LIN {X 0,Y 434.58,Z 409.798,A -85,B 0,C 180,E1 20730.103,E2 20730.103} C_VEL
LIN {X 0,Y 432.075,Z 405.892,A -85,B 0,C 180,E1 20729.227,E2 20729.227} C_VEL
LIN {X 0,Y 431.039,Z 404.203,A -85,B 0,C 180,E1 20728.847,E2 20728.847} C_VEL
LIN {X 0,Y 428.961,Z 400.99,A -85,B 0,C 180,E1 20728.088,E2 20728.088} C_VEL
LIN {X 0,Y 428.028,Z 399.18,A -85,B 0,C 180,E1 20727.7,E2 20727.7} C_VEL
LIN {X 0,Y 425.933,Z 396.363,A -85,B 0,C 180,E1 20726.94,E2 20726.94} C_VEL
LIN {X 0,Y 425.284,Z 394.314,A -85,B 0,C 180,E1 20726.456,E2 20726.456} C_VEL
LIN {X 0,Y 425.267,Z 394.05,A -85,B 0,C 180,E1 20723.516,E2 20723.516} C_VEL
LIN {X 0,Y 425.242,Z 394.017,A -85,B 0,C 180,E1 20719.79,E2 20719.79} C_VEL
LIN {X 0,Y 425.248,Z 394.073,A -85,B 0,C 180,E1 20715.916,E2 20715.916} C_VEL
LIN {X 0,Y 425.277,Z 394.009,A -85,B 0,C 180,E1 20712.353,E2 20712.353} C_VEL
LIN {X 0,Y 425.301,Z 394.055,A -85,B 0,C 180,E1 20708.517,E2 20708.517} C_VEL
LIN {X 0,Y 425.258,Z 394.062,A -85,B 0,C 180,E1 20704.855,E2 20704.855} C_VEL
LIN {X 0,Y 425.247,Z 394.066,A -85,B 0,C 180,E1 20701.077,E2 20701.077} C_VEL
LIN {X 0,Y 425.256,Z 394.066,A -85,B 0,C 180,E1 20697.304,E2 20697.304} C_VEL
LIN {X 0,Y 425.299,Z 394.061,A -85,B 0,C 180,E1 20693.656,E2 20693.656} C_VEL
LIN {X 0,Y 425.291,Z 394.062,A -85,B 0,C 180,E1 20689.844,E2 20689.844} C_VEL
LIN {X 0,Y 425.26,Z 394.069,A -85,B 0,C 180,E1 20686.124,E2 20686.124} C_VEL
LIN {X 0,Y 425.252,Z 394.069,A -85,B 0,C 180,E1 20682.343,E2 20682.343} C_VEL
LIN {X 0,Y 425.266,Z 394.063,A -85,B 0,C 180,E1 20678.6,E2 20678.6} C_VEL
LIN {X 0,Y 425.303,Z 394.058,A -85,B 0,C 180,E1 20674.965,E2 20674.965} C_VEL
LIN {X 0,Y 425.281,Z 394.029,A -85,B 0,C 180,E1 20671.186,E2 20671.186} C_VEL
LIN {X 0,Y 425.255,Z 394.054,A -85,B 0,C 180,E1 20667.574,E2 20667.574} C_VEL
LIN {X 0,Y 425.302,Z 394.194,A -85,B 0,C 180,E1 20664.169,E2 20664.169} C_VEL
LIN {X 0,Y 425.713,Z 395.877,A -85,B 0,C 180,E1 20663.71,E2 20663.71} C_VEL
LIN {X 0,Y 427.779,Z 398.931,A -85,B 0,C 180,E1 20662.848,E2 20662.848} C_VEL
LIN {X 0,Y 430.392,Z 403.77,A -85,B 0,C 180,E1 20661.663,E2 20661.663} C_VEL
LIN {X 0,Y 433.946,Z 410.444,A -85,B 0,C 180,E1 20660.11,E2 20660.11} C_VEL
LIN {X 0,Y 438.166,Z 418.16,A -85,B 0,C 180,E1 20658.391,E2 20658.391} C_VEL
LIN {X 0,Y 445.271,Z 432.655,A -85,B 0,C 180,E1 20655.525,E2 20655.525} C_VEL
LIN {X 0,Y 452.585,Z 448.692,A -85,B 0,C 180,E1 20652.706,E2 20652.706} C_VEL
LIN {X 0,Y 455.691,Z 456.291,A -85,B 0,C 180,E1 20651.502,E2 20651.502} C_VEL
LIN {X 0,Y 454.277,Z 469.929,A -85,B 0,C 180,E1 20650.379,E2 20650.379} C_VEL
LIN {X 0,Y 459.417,Z 502.519,A -85,B 0,C 180,E1 20649.065,E2 20649.065} C_VEL
LIN {X 0,Y 455.217,Z 710.635,A -85,B 0,C 180,E1 20645.736,E2 20645.736} C_VEL
LIN {X 0,Y 454.338,Z 718.35,A -85,B 0,C 180,E1 20645.703,E2 20645.703} C_VEL
LIN {X 0,Y 449.299,Z 738.921,A -85,B 0,C 180,E1 20645.888,E2 20645.888} C_VEL
LIN {X 0,Y 448.519,Z 745.495,A -85,B 0,C 180,E1 20645.816,E2 20645.816} C_VEL
LIN {X 0,Y 447.473,Z 766.05,A -85,B 0,C 180,E1 20645.239,E2 20645.239} C_VEL
LIN {X 0,Y 445.953,Z 785.206,A -85,B 0,C 180,E1 20644.481,E2 20644.481} C_VEL
LIN {X 0,Y 443.922,Z 804.341,A -85,B 0,C 180,E1 20643.492,E2 20643.492} C_VEL
LIN {X 0,Y 441.499,Z 822.584,A -85,B 0,C 180,E1 20642.308,E2 20642.308} C_VEL
LIN {X 0,Y 438.747,Z 839.761,A -85,B 0,C 180,E1 20640.924,E2 20640.924} C_VEL
LIN {X 0,Y 435.749,Z 856.312,A -85,B 0,C 180,E1 20639.315,E2 20639.315} C_VEL
LIN {X 0,Y 432.716,Z 871.672,A -85,B 0,C 180,E1 20637.525,E2 20637.525} C_VEL
LIN {X 0,Y 429.626,Z 886.219,A -85,B 0,C 180,E1 20635.502,E2 20635.502} C_VEL
LIN {X 0,Y 426.599,Z 899.958,A -85,B 0,C 180,E1 20633.189,E2 20633.189} C_VEL
LIN {X 0,Y 424.003,Z 911.448,A -85,B 0,C 180,E1 20630.86,E2 20630.86} C_VEL
LIN {X 0,Y 421.69,Z 922.146,A -85,B 0,C 180,E1 20628.239,E2 20628.239} C_VEL
LIN {X 0,Y 419.815,Z 931.325,A -85,B 0,C 180,E1 20625.471,E2 20625.471} C_VEL
LIN {X 0,Y 418.496,Z 938.657,A -85,B 0,C 180,E1 20622.698,E2 20622.698} C_VEL
LIN {X 0,Y 417.578,Z 944.582,A -85,B 0,C 180,E1 20619.788,E2 20619.788} C_VEL
LIN {X 0,Y 417.042,Z 948.963,A -85,B 0,C 180,E1 20616.747,E2 20616.747} C_VEL
LIN {X 0,Y 416.752,Z 951.583,A -85,B 0,C 180,E1 20613.852,E2 20613.852} C_VEL
LIN {X 0,Y 416.652,Z 952.799,A -85,B 0,C 180,E1 20610.825,E2 20610.825} C_VEL
LIN {X 0,Y 416.68,Z 952.48,A -85,B 0,C 180,E1 20607.8,E2 20607.8} C_VEL
LIN {X 0,Y 416.847,Z 950.752,A -85,B 0,C 180,E1 20604.908,E2 20604.908} C_VEL
LIN {X 0,Y 417.232,Z 947.317,A -85,B 0,C 180,E1 20601.872,E2 20601.872} C_VEL
LIN {X 0,Y 417.879,Z 942.403,A -85,B 0,C 180,E1 20598.965,E2 20598.965} C_VEL
LIN {X 0,Y 418.936,Z 936.141,A -85,B 0,C 180,E1 20596.192,E2 20596.192} C_VEL
LIN {X 0,Y 420.522,Z 927.732,A -85,B 0,C 180,E1 20593.28,E2 20593.28} C_VEL
LIN {X 0,Y 422.54,Z 918.272,A -85,B 0,C 180,E1 20590.653,E2 20590.653} C_VEL
LIN {X 0,Y 424.926,Z 907.438,A -85,B 0,C 180,E1 20588.175,E2 20588.175} C_VEL
LIN {X 0,Y 427.856,Z 894.306,A -85,B 0,C 180,E1 20585.714,E2 20585.714} C_VEL
LIN {X 0,Y 430.749,Z 880.956,A -85,B 0,C 180,E1 20583.636,E2 20583.636} C_VEL
LIN {X 0,Y 433.918,Z 865.8,A -85,B 0,C 180,E1 20581.661,E2 20581.661} C_VEL
LIN {X 0,Y 436.855,Z 850.568,A -85,B 0,C 180,E1 20579.993,E2 20579.993} C_VEL
LIN {X 0,Y 439.776,Z 833.812,A -85,B 0,C 180,E1 20578.471,E2 20578.471} C_VEL
LIN {X 0,Y 442.262,Z 817.144,A -85,B 0,C 180,E1 20577.224,E2 20577.224} C_VEL
LIN {X 0,Y 444.629,Z 798.35,A -85,B 0,C 180,E1 20576.077,E2 20576.077} C_VEL
LIN {X 0,Y 446.547,Z 779.048,A -85,B 0,C 180,E1 20575.153,E2 20575.153} C_VEL
LIN {X 0,Y 447.929,Z 759.118,A -85,B 0,C 180,E1 20574.45,E2 20574.45} C_VEL
LIN {X 0,Y 448.685,Z 739.004,A -85,B 0,C 180,E1 20573.963,E2 20573.963} C_VEL
LIN {X 0,Y 453.726,Z 503.211,A -85,B 0,C 180,E1 20570.137,E2 20570.137} C_VEL
LIN {X 0,Y 448.407,Z 469.022,A -85,B 0,C 180,E1 20568.698,E2 20568.698} C_VEL
LIN {X 0,Y 449.38,Z 459.9,A -85,B 0,C 180,E1 20567.905,E2 20567.905} C_VEL
LIN {X 0,Y 442.411,Z 443.705,A -85,B 0,C 180,E1 20565.16,E2 20565.16} C_VEL
LIN {X 0,Y 435.054,Z 428.114,A -85,B 0,C 180,E1 20562.151,E2 20562.151} C_VEL
LIN {X 0,Y 429.426,Z 417.514,A -85,B 0,C 180,E1 20559.815,E2 20559.815} C_VEL
LIN {X 0,Y 425.397,Z 409.839,A -85,B 0,C 180,E1 20558.011,E2 20558.011} C_VEL
LIN {X 0,Y 423.204,Z 405.593,A -85,B 0,C 180,E1 20556.971,E2 20556.971} C_VEL
LIN {X 0,Y 420.658,Z 401.587,A -85,B 0,C 180,E1 20555.853,E2 20555.853} C_VEL
LIN {X 0,Y 420.071,Z 400.09,A -85,B 0,C 180,E1 20555.505,E2 20555.505} C_VEL
LIN {X 0,Y 417.86,Z 397.077,A -85,B 0,C 180,E1 20554.548,E2 20554.548} C_VEL
LIN {X 0,Y 417.352,Z 395.211,A -85,B 0,C 180,E1 20554.012,E2 20554.012} C_VEL
LIN {X 0,Y 417.314,Z 395.002,A -85,B 0,C 180,E1 20550.209,E2 20550.209} C_VEL
LIN {X 0,Y 417.334,Z 395.057,A -85,B 0,C 180,E1 20546.464,E2 20546.464} C_VEL
LIN {X 0,Y 417.363,Z 395.047,A -85,B 0,C 180,E1 20542.688,E2 20542.688} C_VEL
LIN {X 0,Y 417.363,Z 395.045,A -85,B 0,C 180,E1 20538.863,E2 20538.863} C_VEL
LIN {X 0,Y 417.33,Z 395.047,A -85,B 0,C 180,E1 20535.087,E2 20535.087} C_VEL
LIN {X 0,Y 417.315,Z 395.047,A -85,B 0,C 180,E1 20531.331,E2 20531.331} C_VEL
LIN {X 0,Y 417.316,Z 395.047,A -85,B 0,C 180,E1 20527.434,E2 20527.434} C_VEL
LIN {X 0,Y 417.341,Z 395.046,A -85,B 0,C 180,E1 20523.709,E2 20523.709} C_VEL
LIN {X 0,Y 417.373,Z 395.042,A -85,B 0,C 180,E1 20519.863,E2 20519.863} C_VEL
LIN {X 0,Y 417.344,Z 395.046,A -85,B 0,C 180,E1 20516.016,E2 20516.016} C_VEL
LIN {X 0,Y 417.313,Z 395.049,A -85,B 0,C 180,E1 20512.428,E2 20512.428} C_VEL
LIN {X 0,Y 417.305,Z 395.017,A -85,B 0,C 180,E1 20508.512,E2 20508.512} C_VEL
LIN {X 0,Y 417.322,Z 395.033,A -85,B 0,C 180,E1 20504.72,E2 20504.72} C_VEL
LIN {X 0,Y 417.351,Z 394.998,A -85,B 0,C 180,E1 20500.985,E2 20500.985} C_VEL
LIN {X 0,Y 417.347,Z 395.058,A -85,B 0,C 180,E1 20497.164,E2 20497.164} C_VEL
LIN {X 0,Y 417.366,Z 395.312,A -85,B 0,C 180,E1 20495.29,E2 20495.29} C_VEL
LIN {X 0,Y 418.54,Z 398.331,A -85,B 0,C 180,E1 20494.533,E2 20494.533} C_VEL
LIN {X 0,Y 420.656,Z 400.699,A -85,B 0,C 180,E1 20493.762,E2 20493.762} C_VEL
LIN {X 0,Y 422.743,Z 404.706,A -85,B 0,C 180,E1 20492.841,E2 20492.841} C_VEL
LIN {X 0,Y 424.136,Z 406.649,A -85,B 0,C 180,E1 20492.329,E2 20492.329} C_VEL
LIN {X 0,Y 426.47,Z 410.53,A -85,B 0,C 180,E1 20491.428,E2 20491.428} C_VEL
LIN {X 0,Y 432.8,Z 420.951,A -85,B 0,C 180,E1 20489.146,E2 20489.146} C_VEL
LIN {X 0,Y 441.671,Z 436.817,A -85,B 0,C 180,E1 20486.159,E2 20486.159} C_VEL
LIN {X 0,Y 449.883,Z 452.515,A -85,B 0,C 180,E1 20483.567,E2 20483.567} C_VEL
LIN {X 0,Y 456.994,Z 467.077,A -85,B 0,C 180,E1 20481.485,E2 20481.485} C_VEL
LIN {X 0,Y 457.833,Z 473.685,A -85,B 0,C 180,E1 20481.224,E2 20481.224} C_VEL
LIN {X 0,Y 460.335,Z 501.186,A -85,B 0,C 180,E1 20480.281,E2 20480.281} C_VEL
LIN {X 0,Y 453.618,Z 693.847,A -85,B 0,C 180,E1 20476.651,E2 20476.651} C_VEL
LIN {X 0,Y 449.66,Z 808.124,A -85,B 0,C 180,E1 20474.468,E2 20474.468} C_VEL
LIN {X 0,Y 447.866,Z 831.918,A -85,B 0,C 180,E1 20473.815,E2 20473.815} C_VEL
LIN {X 0,Y 445.684,Z 855.225,A -85,B 0,C 180,E1 20472.957,E2 20472.957} C_VEL
LIN {X 0,Y 443.239,Z 877.694,A -85,B 0,C 180,E1 20471.891,E2 20471.891} C_VEL
LIN {X 0,Y 440.54,Z 899.902,A -85,B 0,C 180,E1 20470.595,E2 20470.595} C_VEL
LIN {X 0,Y 437.684,Z 921.743,A -85,B 0,C 180,E1 20469.088,E2 20469.088} C_VEL
LIN {X 0,Y 434.294,Z 946.962,A -85,B 0,C 180,E1 20467.017,E2 20467.017} C_VEL
LIN {X 0,Y 431.456,Z 967.018,A -85,B 0,C 180,E1 20465.08,E2 20465.08} C_VEL
LIN {X 0,Y 428.702,Z 986.424,A -85,B 0,C 180,E1 20462.917,E2 20462.917} C_VEL
LIN {X 0,Y 426.391,Z 1002.164,A -85,B 0,C 180,E1 20460.881,E2 20460.881} C_VEL
LIN {X 0,Y 423.873,Z 1019.48,A -85,B 0,C 180,E1 20458.303,E2 20458.303} C_VEL
LIN {X 0,Y 421.964,Z 1032.879,A -85,B 0,C 180,E1 20456,E2 20456} C_VEL
LIN {X 0,Y 420.036,Z 1047.189,A -85,B 0,C 180,E1 20453.127,E2 20453.127} C_VEL
LIN {X 0,Y 418.712,Z 1058.007,A -85,B 0,C 180,E1 20450.599,E2 20450.599} C_VEL
LIN {X 0,Y 417.617,Z 1067.985,A -85,B 0,C 180,E1 20447.846,E2 20447.846} C_VEL
LIN {X 0,Y 416.918,Z 1074.78,A -85,B 0,C 180,E1 20445.405,E2 20445.405} C_VEL
LIN {X 0,Y 416.349,Z 1081.771,A -85,B 0,C 180,E1 20442.341,E2 20442.341} C_VEL
LIN {X 0,Y 416.056,Z 1087.049,A -85,B 0,C 180,E1 20439.266,E2 20439.266} C_VEL
LIN {X 0,Y 415.944,Z 1090.757,A -85,B 0,C 180,E1 20436.349,E2 20436.349} C_VEL
LIN {X 0,Y 415.887,Z 1093.052,A -85,B 0,C 180,E1 20433.308,E2 20433.308} C_VEL
LIN {X 0,Y 415.885,Z 1093.893,A -85,B 0,C 180,E1 20430.689,E2 20430.689} C_VEL
LIN {X 0,Y 415.907,Z 1093.46,A -85,B 0,C 180,E1 20427.52,E2 20427.52} C_VEL
LIN {X 0,Y 415.919,Z 1091.726,A -85,B 0,C 180,E1 20424.759,E2 20424.759} C_VEL
LIN {X 0,Y 416.011,Z 1088.494,A -85,B 0,C 180,E1 20421.709,E2 20421.709} C_VEL
LIN {X 0,Y 416.22,Z 1083.572,A -85,B 0,C 180,E1 20418.639,E2 20418.639} C_VEL
LIN {X 0,Y 416.691,Z 1077.166,A -85,B 0,C 180,E1 20415.549,E2 20415.549} C_VEL
LIN {X 0,Y 417.378,Z 1070.114,A -85,B 0,C 180,E1 20412.863,E2 20412.863} C_VEL
LIN {X 0,Y 418.091,Z 1063.479,A -85,B 0,C 180,E1 20410.844,E2 20410.844} C_VEL
LIN {X 0,Y 419.416,Z 1052.381,A -85,B 0,C 180,E1 20408.02,E2 20408.02} C_VEL
LIN {X 0,Y 421.062,Z 1039.618,A -85,B 0,C 180,E1 20405.296,E2 20405.296} C_VEL
LIN {X 0,Y 423.006,Z 1025.637,A -85,B 0,C 180,E1 20402.706,E2 20402.706} C_VEL
LIN {X 0,Y 425.227,Z 1010.135,A -85,B 0,C 180,E1 20400.255,E2 20400.255} C_VEL
LIN {X 0,Y 427.878,Z 991.988,A -85,B 0,C 180,E1 20397.769,E2 20397.769} C_VEL
LIN {X 0,Y 430.415,Z 974.526,A -85,B 0,C 180,E1 20395.713,E2 20395.713} C_VEL
LIN {X 0,Y 433.185,Z 954.615,A -85,B 0,C 180,E1 20393.692,E2 20393.692} C_VEL
LIN {X 0,Y 436.1,Z 933.629,A -85,B 0,C 180,E1 20391.85,E2 20391.85} C_VEL
LIN {X 0,Y 438.987,Z 911.918,A -85,B 0,C 180,E1 20390.206,E2 20390.206} C_VEL
LIN {X 0,Y 441.873,Z 888.896,A -85,B 0,C 180,E1 20388.73,E2 20388.73} C_VEL
LIN {X 0,Y 444.571,Z 866.255,A -85,B 0,C 180,E1 20387.534,E2 20387.534} C_VEL
LIN {X 0,Y 446.832,Z 843.574,A -85,B 0,C 180,E1 20386.587,E2 20386.587} C_VEL
LIN {X 0,Y 448.875,Z 819.392,A -85,B 0,C 180,E1 20385.817,E2 20385.817} C_VEL
LIN {X 0,Y 450.202,Z 795.783,A -85,B 0,C 180,E1 20385.274,E2 20385.274} C_VEL
LIN {X 0,Y 457.399,Z 585.058,A -85,B 0,C 180,E1 20381.292,E2 20381.292} C_VEL
LIN {X 0,Y 460.227,Z 498.698,A -85,B 0,C 180,E1 20379.656,E2 20379.656} C_VEL
LIN {X 0,Y 457.045,Z 467.185,A -85,B 0,C 180,E1 20378.53,E2 20378.53} C_VEL
LIN {X 0,Y 450.952,Z 454.7,A -85,B 0,C 180,E1 20376.773,E2 20376.773} C_VEL
LIN {X 0,Y 442.418,Z 438.137,A -85,B 0,C 180,E1 20374.088,E2 20374.088} C_VEL
LIN {X 0,Y 434.866,Z 424.794,A -85,B 0,C 180,E1 20371.616,E2 20371.616} C_VEL
LIN {X 0,Y 429.521,Z 415.576,A -85,B 0,C 180,E1 20369.724,E2 20369.724} C_VEL
LIN {X 0,Y 426.409,Z 410.466,A -85,B 0,C 180,E1 20368.577,E2 20368.577} C_VEL
LIN {X 0,Y 424.093,Z 406.55,A -85,B 0,C 180,E1 20367.674,E2 20367.674} C_VEL
LIN {X 0,Y 420.948,Z 401.548,A -85,B 0,C 180,E1 20366.43,E2 20366.43} C_VEL
LIN {X 0,Y 420.214,Z 400.277,A -85,B 0,C 180,E1 20366.115,E2 20366.115} C_VEL
LIN {X 0,Y 417.919,Z 397.123,A -85,B 0,C 180,E1 20365.205,E2 20365.205} C_VEL
LIN {X 0,Y 417.385,Z 395.389,A -85,B 0,C 180,E1 20364.781,E2 20364.781} C_VEL
LIN {X 0,Y 417.322,Z 395.035,A -85,B 0,C 180,E1 20363.585,E2 20363.585} C_VEL
LIN {X 0,Y 417.302,Z 395.003,A -85,B 0,C 180,E1 20359.891,E2 20359.891} C_VEL
LIN {X 0,Y 417.311,Z 395.062,A -85,B 0,C 180,E1 20355.993,E2 20355.993} C_VEL
LIN {X 0,Y 417.334,Z 394.996,A -85,B 0,C 180,E1 20352.311,E2 20352.311} C_VEL
LIN {X 0,Y 417.36,Z 395.044,A -85,B 0,C 180,E1 20348.541,E2 20348.541} C_VEL
LIN {X 0,Y 417.322,Z 395.049,A -85,B 0,C 180,E1 20344.81,E2 20344.81} C_VEL
LIN {X 0,Y 417.308,Z 395.054,A -85,B 0,C 180,E1 20341.098,E2 20341.098} C_VEL
LIN {X 0,Y 417.315,Z 395.054,A -85,B 0,C 180,E1 20337.253,E2 20337.253} C_VEL
LIN {X 0,Y 417.346,Z 395.05,A -85,B 0,C 180,E1 20333.534,E2 20333.534} C_VEL
LIN {X 0,Y 417.356,Z 395.049,A -85,B 0,C 180,E1 20329.788,E2 20329.788} C_VEL
LIN {X 0,Y 417.329,Z 395.054,A -85,B 0,C 180,E1 20325.996,E2 20325.996} C_VEL
LIN {X 0,Y 417.313,Z 395.056,A -85,B 0,C 180,E1 20322.284,E2 20322.284} C_VEL
LIN {X 0,Y 417.317,Z 395.051,A -85,B 0,C 180,E1 20318.377,E2 20318.377} C_VEL
LIN {X 0,Y 417.354,Z 395.046,A -85,B 0,C 180,E1 20314.758,E2 20314.758} C_VEL
LIN {X 0,Y 417.366,Z 395.007,A -85,B 0,C 180,E1 20310.901,E2 20310.901} C_VEL
LIN {X 0,Y 417.341,Z 395.056,A -85,B 0,C 180,E1 20307.054,E2 20307.054} C_VEL
LIN {X 0,Y 417.358,Z 395.319,A -85,B 0,C 180,E1 20305.792,E2 20305.792} C_VEL
LIN {X 0,Y 418.786,Z 398.696,A -85,B 0,C 180,E1 20304.873,E2 20304.873} C_VEL
LIN {X 0,Y 420.403,Z 400.841,A -85,B 0,C 180,E1 20304.192,E2 20304.192} C_VEL
LIN {X 0,Y 422.422,Z 404.634,A -85,B 0,C 180,E1 20303.213,E2 20303.213} C_VEL
LIN {X 0,Y 423.366,Z 406.161,A -85,B 0,C 180,E1 20302.8,E2 20302.8} C_VEL
LIN {X 0,Y 428.328,Z 415.161,A -85,B 0,C 180,E1 20300.584,E2 20300.584} C_VEL
LIN {X 0,Y 435.468,Z 429.169,A -85,B 0,C 180,E1 20297.542,E2 20297.542} C_VEL
LIN {X 0,Y 442.295,Z 443.512,A -85,B 0,C 180,E1 20294.778,E2 20294.778} C_VEL
LIN {X 0,Y 449.359,Z 459.915,A -85,B 0,C 180,E1 20291.997,E2 20291.997} C_VEL
LIN {X 0,Y 448.421,Z 469.809,A -85,B 0,C 180,E1 20291.165,E2 20291.165} C_VEL
LIN {X 0,Y 453.706,Z 504.187,A -85,B 0,C 180,E1 20289.75,E2 20289.75} C_VEL
LIN {X 0,Y 449.05,Z 719.472,A -85,B 0,C 180,E1 20286.271,E2 20286.271} C_VEL
LIN {X 0,Y 448.519,Z 745.495,A -85,B 0,C 180,E1 20285.816,E2 20285.816} C_VEL
LIN {X 0,Y 447.42,Z 753.146,A -85,B 0,C 180,E1 20285.716,E2 20285.716} C_VEL
LIN {X 0,Y 441.65,Z 772.397,A -85,B 0,C 180,E1 20285.632,E2 20285.632} C_VEL
LIN {X 0,Y 440.416,Z 779.867,A -85,B 0,C 180,E1 20285.414,E2 20285.414} C_VEL
LIN {X 0,Y 438.486,Z 798.51,A -85,B 0,C 180,E1 20284.517,E2 20284.517} C_VEL
LIN {X 0,Y 436.082,Z 817.076,A -85,B 0,C 180,E1 20283.386,E2 20283.386} C_VEL
LIN {X 0,Y 433.467,Z 834.043,A -85,B 0,C 180,E1 20282.12,E2 20282.12} C_VEL
LIN {X 0,Y 430.395,Z 850.896,A -85,B 0,C 180,E1 20280.582,E2 20280.582} C_VEL
LIN {X 0,Y 427.193,Z 866.851,A -85,B 0,C 180,E1 20278.826,E2 20278.826} C_VEL
LIN {X 0,Y 423.796,Z 882.328,A -85,B 0,C 180,E1 20276.784,E2 20276.784} C_VEL
LIN {X 0,Y 420.819,Z 895.424,A -85,B 0,C 180,E1 20274.72,E2 20274.72} C_VEL
LIN {X 0,Y 417.718,Z 908.587,A -85,B 0,C 180,E1 20272.222,E2 20272.222} C_VEL
LIN {X 0,Y 415.128,Z 919.661,A -85,B 0,C 180,E1 20269.653,E2 20269.653} C_VEL
LIN {X 0,Y 412.992,Z 929.053,A -85,B 0,C 180,E1 20267,E2 20267} C_VEL
LIN {X 0,Y 411.301,Z 937.38,A -85,B 0,C 180,E1 20264.07,E2 20264.07} C_VEL
LIN {X 0,Y 410.1,Z 943.929,A -85,B 0,C 180,E1 20261.105,E2 20261.105} C_VEL
LIN {X 0,Y 409.399,Z 948.784,A -85,B 0,C 180,E1 20258.143,E2 20258.143} C_VEL
LIN {X 0,Y 408.984,Z 952.185,A -85,B 0,C 180,E1 20255.049,E2 20255.049} C_VEL
LIN {X 0,Y 408.796,Z 953.928,A -85,B 0,C 180,E1 20251.962,E2 20251.962} C_VEL
LIN {X 0,Y 408.769,Z 954.159,A -85,B 0,C 180,E1 20249.019,E2 20249.019} C_VEL
LIN {X 0,Y 408.885,Z 952.93,A -85,B 0,C 180,E1 20245.933,E2 20245.933} C_VEL
LIN {X 0,Y 409.209,Z 950.307,A -85,B 0,C 180,E1 20242.983,E2 20242.983} C_VEL
LIN {X 0,Y 409.8,Z 945.93,A -85,B 0,C 180,E1 20239.882,E2 20239.882} C_VEL
LIN {X 0,Y 410.88,Z 939.65,A -85,B 0,C 180,E1 20236.752,E2 20236.752} C_VEL
LIN {X 0,Y 412.407,Z 931.865,A -85,B 0,C 180,E1 20233.811,E2 20233.811} C_VEL
LIN {X 0,Y 414.447,Z 922.609,A -85,B 0,C 180,E1 20231.034,E2 20231.034} C_VEL
LIN {X 0,Y 416.85,Z 912.156,A -85,B 0,C 180,E1 20228.47,E2 20228.47} C_VEL
LIN {X 0,Y 419.633,Z 900.525,A -85,B 0,C 180,E1 20226.105,E2 20226.105} C_VEL
LIN {X 0,Y 422.657,Z 887.546,A -85,B 0,C 180,E1 20223.895,E2 20223.895} C_VEL
LIN {X 0,Y 425.901,Z 873.003,A -85,B 0,C 180,E1 20221.844,E2 20221.844} C_VEL
LIN {X 0,Y 429.063,Z 857.77,A -85,B 0,C 180,E1 20220.043,E2 20220.043} C_VEL
LIN {X 0,Y 432.227,Z 841.142,A -85,B 0,C 180,E1 20218.402,E2 20218.402} C_VEL
LIN {X 0,Y 435.105,Z 823.982,A -85,B 0,C 180,E1 20217.001,E2 20217.001} C_VEL
LIN {X 0,Y 437.658,Z 805.649,A -85,B 0,C 180,E1 20215.794,E2 20215.794} C_VEL
LIN {X 0,Y 439.77,Z 786.819,A -85,B 0,C 180,E1 20214.805,E2 20214.805} C_VEL
LIN {X 0,Y 441.4,Z 767.446,A -85,B 0,C 180,E1 20214.022,E2 20214.022} C_VEL
LIN {X 0,Y 442.512,Z 746.743,A -85,B 0,C 180,E1 20213.43,E2 20213.43} C_VEL
LIN {X 0,Y 443.439,Z 704.039,A -85,B 0,C 180,E1 20212.699,E2 20212.699} C_VEL
LIN {X 0,Y 448.094,Z 504.78,A -85,B 0,C 180,E1 20209.433,E2 20209.433} C_VEL
LIN {X 0,Y 442.67,Z 468.634,A -85,B 0,C 180,E1 20207.868,E2 20207.868} C_VEL
LIN {X 0,Y 443.149,Z 463.892,A -85,B 0,C 180,E1 20207.439,E2 20207.439} C_VEL
LIN {X 0,Y 436.539,Z 448.439,A -85,B 0,C 180,E1 20204.762,E2 20204.762} C_VEL
LIN {X 0,Y 429.651,Z 433.661,A -85,B 0,C 180,E1 20201.867,E2 20201.867} C_VEL
LIN {X 0,Y 424.37,Z 423.517,A -85,B 0,C 180,E1 20199.606,E2 20199.606} C_VEL
LIN {X 0,Y 420.177,Z 415.604,A -85,B 0,C 180,E1 20197.703,E2 20197.703} C_VEL
LIN {X 0,Y 417.481,Z 410.731,A -85,B 0,C 180,E1 20196.439,E2 20196.439} C_VEL
LIN {X 0,Y 415.385,Z 406.622,A -85,B 0,C 180,E1 20195.374,E2 20195.374} C_VEL
LIN {X 0,Y 412.843,Z 402.739,A -85,B 0,C 180,E1 20194.186,E2 20194.186} C_VEL
LIN {X 0,Y 412.109,Z 401.106,A -85,B 0,C 180,E1 20193.753,E2 20193.753} C_VEL
LIN {X 0,Y 409.801,Z 397.754,A -85,B 0,C 180,E1 20192.63,E2 20192.63} C_VEL
LIN {X 0,Y 409.411,Z 396.228,A -85,B 0,C 180,E1 20192.168,E2 20192.168} C_VEL
LIN {X 0,Y 409.402,Z 396.001,A -85,B 0,C 180,E1 20188.745,E2 20188.745} C_VEL
LIN {X 0,Y 409.429,Z 396.033,A -85,B 0,C 180,E1 20184.992,E2 20184.992} C_VEL
LIN {X 0,Y 409.407,Z 396.039,A -85,B 0,C 180,E1 20181.19,E2 20181.19} C_VEL
LIN {X 0,Y 409.382,Z 396.045,A -85,B 0,C 180,E1 20177.483,E2 20177.483} C_VEL
LIN {X 0,Y 409.379,Z 396.049,A -85,B 0,C 180,E1 20173.561,E2 20173.561} C_VEL
LIN {X 0,Y 409.388,Z 396.049,A -85,B 0,C 180,E1 20169.702,E2 20169.702} C_VEL
LIN {X 0,Y 409.412,Z 396.046,A -85,B 0,C 180,E1 20165.888,E2 20165.888} C_VEL
LIN {X 0,Y 409.426,Z 396.046,A -85,B 0,C 180,E1 20161.96,E2 20161.96} C_VEL
LIN {X 0,Y 409.402,Z 396.049,A -85,B 0,C 180,E1 20158.181,E2 20158.181} C_VEL
LIN {X 0,Y 409.38,Z 396.053,A -85,B 0,C 180,E1 20154.394,E2 20154.394} C_VEL
LIN {X 0,Y 409.373,Z 396.055,A -85,B 0,C 180,E1 20150.582,E2 20150.582} C_VEL
LIN {X 0,Y 409.375,Z 395.982,A -85,B 0,C 180,E1 20146.728,E2 20146.728} C_VEL
LIN {X 0,Y 409.421,Z 396.038,A -85,B 0,C 180,E1 20143.106,E2 20143.106} C_VEL
LIN {X 0,Y 409.416,Z 395.994,A -85,B 0,C 180,E1 20139.112,E2 20139.112} C_VEL
LIN {X 0,Y 409.405,Z 396.127,A -85,B 0,C 180,E1 20137.303,E2 20137.303} C_VEL
LIN {X 0,Y 409.701,Z 397.34,A -85,B 0,C 180,E1 20136.865,E2 20136.865} C_VEL
LIN {X 0,Y 411.326,Z 400.338,A -85,B 0,C 180,E1 20136.05,E2 20136.05} C_VEL
LIN {X 0,Y 413.01,Z 402.188,A -85,B 0,C 180,E1 20135.393,E2 20135.393} C_VEL
LIN {X 0,Y 415,Z 405.922,A -85,B 0,C 180,E1 20134.453,E2 20134.453} C_VEL
LIN {X 0,Y 416.405,Z 407.776,A -85,B 0,C 180,E1 20133.902,E2 20133.902} C_VEL
LIN {X 0,Y 418.901,Z 411.842,A -85,B 0,C 180,E1 20132.878,E2 20132.878} C_VEL
LIN {X 0,Y 423.187,Z 419.101,A -85,B 0,C 180,E1 20131.185,E2 20131.185} C_VEL
LIN {X 0,Y 428.11,Z 427.224,A -85,B 0,C 180,E1 20129.394,E2 20129.394} C_VEL
LIN {X 0,Y 436.871,Z 443.057,A -85,B 0,C 180,E1 20126.368,E2 20126.368} C_VEL
LIN {X 0,Y 445.299,Z 459.436,A -85,B 0,C 180,E1 20123.646,E2 20123.646} C_VEL
LIN {X 0,Y 449.173,Z 467.259,A -85,B 0,C 180,E1 20122.517,E2 20122.517} C_VEL
LIN {X 0,Y 451.921,Z 472.038,A -85,B 0,C 180,E1 20122.033,E2 20122.033} C_VEL
LIN {X 0,Y 454.613,Z 502.552,A -85,B 0,C 180,E1 20120.966,E2 20120.966} C_VEL
LIN {X 0,Y 447.586,Z 693.963,A -85,B 0,C 180,E1 20117.321,E2 20117.321} C_VEL
LIN {X 0,Y 443.446,Z 807.078,A -85,B 0,C 180,E1 20115.132,E2 20115.132} C_VEL
LIN {X 0,Y 441.597,Z 830.727,A -85,B 0,C 180,E1 20114.479,E2 20114.479} C_VEL
LIN {X 0,Y 439.372,Z 853.398,A -85,B 0,C 180,E1 20113.643,E2 20113.643} C_VEL
LIN {X 0,Y 436.797,Z 875.51,A -85,B 0,C 180,E1 20112.593,E2 20112.593} C_VEL
LIN {X 0,Y 433.841,Z 898.594,A -85,B 0,C 180,E1 20111.234,E2 20111.234} C_VEL
LIN {X 0,Y 430.878,Z 919.893,A -85,B 0,C 180,E1 20109.74,E2 20109.74} C_VEL
LIN {X 0,Y 427.688,Z 941.372,A -85,B 0,C 180,E1 20107.941,E2 20107.941} C_VEL
LIN {X 0,Y 424.335,Z 963.804,A -85,B 0,C 180,E1 20105.758,E2 20105.758} C_VEL
LIN {X 0,Y 421.496,Z 982.967,A -85,B 0,C 180,E1 20103.631,E2 20103.631} C_VEL
LIN {X 0,Y 418.833,Z 1000.458,A -85,B 0,C 180,E1 20101.361,E2 20101.361} C_VEL
LIN {X 0,Y 416.316,Z 1017.169,A -85,B 0,C 180,E1 20098.865,E2 20098.865} C_VEL
LIN {X 0,Y 414.261,Z 1031.15,A -85,B 0,C 180,E1 20096.436,E2 20096.436} C_VEL
LIN {X 0,Y 412.277,Z 1045.486,A -85,B 0,C 180,E1 20093.549,E2 20093.549} C_VEL
LIN {X 0,Y 410.882,Z 1056.426,A -85,B 0,C 180,E1 20090.96,E2 20090.96} C_VEL
LIN {X 0,Y 409.623,Z 1067.585,A -85,B 0,C 180,E1 20087.834,E2 20087.834} C_VEL
LIN {X 0,Y 408.853,Z 1075.501,A -85,B 0,C 180,E1 20085.169,E2 20085.169} C_VEL
LIN {X 0,Y 408.37,Z 1082.016,A -85,B 0,C 180,E1 20082.443,E2 20082.443} C_VEL
LIN {X 0,Y 408.066,Z 1087.049,A -85,B 0,C 180,E1 20079.449,E2 20079.449} C_VEL
LIN {X 0,Y 407.949,Z 1090.757,A -85,B 0,C 180,E1 20076.474,E2 20076.474} C_VEL
LIN {X 0,Y 407.888,Z 1093.051,A -85,B 0,C 180,E1 20073.373,E2 20073.373} C_VEL
LIN {X 0,Y 407.885,Z 1093.893,A -85,B 0,C 180,E1 20070.702,E2 20070.702} C_VEL
LIN {X 0,Y 407.905,Z 1093.459,A -85,B 0,C 180,E1 20067.471,E2 20067.471} C_VEL
LIN {X 0,Y 407.92,Z 1091.726,A -85,B 0,C 180,E1 20064.656,E2 20064.656} C_VEL
LIN {X 0,Y 408.022,Z 1088.494,A -85,B 0,C 180,E1 20061.545,E2 20061.545} C_VEL
LIN {X 0,Y 408.236,Z 1083.826,A -85,B 0,C 180,E1 20058.557,E2 20058.557} C_VEL
LIN {X 0,Y 408.564,Z 1079.142,A -85,B 0,C 180,E1 20056.268,E2 20056.268} C_VEL
LIN {X 0,Y 409.234,Z 1071.465,A -85,B 0,C 180,E1 20053.39,E2 20053.39} C_VEL
LIN {X 0,Y 410.227,Z 1061.879,A -85,B 0,C 180,E1 20050.493,E2 20050.493} C_VEL
LIN {X 0,Y 411.62,Z 1050.533,A -85,B 0,C 180,E1 20047.581,E2 20047.581} C_VEL
LIN {X 0,Y 413.267,Z 1038.332,A -85,B 0,C 180,E1 20044.951,E2 20044.951} C_VEL
LIN {X 0,Y 415.408,Z 1023.364,A -85,B 0,C 180,E1 20042.164,E2 20042.164} C_VEL
LIN {X 0,Y 417.625,Z 1008.565,A -85,B 0,C 180,E1 20039.801,E2 20039.801} C_VEL
LIN {X 0,Y 420.419,Z 989.984,A -85,B 0,C 180,E1 20037.245,E2 20037.245} C_VEL
LIN {X 0,Y 423.193,Z 971.638,A -85,B 0,C 180,E1 20035.068,E2 20035.068} C_VEL
LIN {X 0,Y 426.521,Z 949.232,A -85,B 0,C 180,E1 20032.785,E2 20032.785} C_VEL
LIN {X 0,Y 429.673,Z 927.909,A -85,B 0,C 180,E1 20030.903,E2 20030.903} C_VEL
LIN {X 0,Y 432.814,Z 906.185,A -85,B 0,C 180,E1 20029.263,E2 20029.263} C_VEL
LIN {X 0,Y 435.658,Z 884.753,A -85,B 0,C 180,E1 20027.92,E2 20027.92} C_VEL
LIN {X 0,Y 438.505,Z 861.181,A -85,B 0,C 180,E1 20026.704,E2 20026.704} C_VEL
LIN {X 0,Y 440.885,Z 838.4,A -85,B 0,C 180,E1 20025.772,E2 20025.772} C_VEL
LIN {X 0,Y 442.892,Z 814.758,A -85,B 0,C 180,E1 20025.062,E2 20025.062} C_VEL
LIN {X 0,Y 444.272,Z 787.562,A -85,B 0,C 180,E1 20024.468,E2 20024.468} C_VEL
LIN {X 0,Y 451.808,Z 578.498,A -85,B 0,C 180,E1 20020.471,E2 20020.471} C_VEL
LIN {X 0,Y 454.498,Z 500.048,A -85,B 0,C 180,E1 20018.969,E2 20018.969} C_VEL
LIN {X 0,Y 451.663,Z 471.26,A -85,B 0,C 180,E1 20017.921,E2 20017.921} C_VEL
LIN {X 0,Y 447.991,Z 465.17,A -85,B 0,C 180,E1 20017.217,E2 20017.217} C_VEL
LIN {X 0,Y 439.853,Z 448.684,A -85,B 0,C 180,E1 20014.625,E2 20014.625} C_VEL
LIN {X 0,Y 430.757,Z 431.859,A -85,B 0,C 180,E1 20011.562,E2 20011.562} C_VEL
LIN {X 0,Y 424.485,Z 421.293,A -85,B 0,C 180,E1 20009.336,E2 20009.336} C_VEL
LIN {X 0,Y 421.786,Z 416.708,A -85,B 0,C 180,E1 20008.301,E2 20008.301} C_VEL
LIN {X 0,Y 418.469,Z 411.335,A -85,B 0,C 180,E1 20006.998,E2 20006.998} C_VEL
LIN {X 0,Y 415.639,Z 406.619,A -85,B 0,C 180,E1 20005.811,E2 20005.811} C_VEL
LIN {X 0,Y 413.433,Z 403.331,A -85,B 0,C 180,E1 20004.885,E2 20004.885} C_VEL
LIN {X 0,Y 412.661,Z 401.574,A -85,B 0,C 180,E1 20004.476,E2 20004.476} C_VEL
LIN {X 0,Y 410.345,Z 398.946,A -85,B 0,C 180,E1 20003.553,E2 20003.553} C_VEL
LIN {X 0,Y 409.436,Z 396.256,A -85,B 0,C 180,E1 20002.847,E2 20002.847} C_VEL
LIN {X 0,Y 409.39,Z 395.986,A -85,B 0,C 180,E1 19999.251,E2 19999.251} C_VEL
LIN {X 0,Y 409.369,Z 396.033,A -85,B 0,C 180,E1 19995.585,E2 19995.585} C_VEL
LIN {X 0,Y 409.364,Z 395.996,A -85,B 0,C 180,E1 19991.639,E2 19991.639} C_VEL
LIN {X 0,Y 409.38,Z 396.032,A -85,B 0,C 180,E1 19987.861,E2 19987.861} C_VEL
LIN {X 0,Y 409.415,Z 396.029,A -85,B 0,C 180,E1 19984.201,E2 19984.201} C_VEL
LIN {X 0,Y 409.413,Z 396.031,A -85,B 0,C 180,E1 19980.279,E2 19980.279} C_VEL
LIN {X 0,Y 409.383,Z 396.036,A -85,B 0,C 180,E1 19976.499,E2 19976.499} C_VEL
LIN {X 0,Y 409.368,Z 396.036,A -85,B 0,C 180,E1 19972.703,E2 19972.703} C_VEL
LIN {X 0,Y 409.378,Z 396.035,A -85,B 0,C 180,E1 19968.875,E2 19968.875} C_VEL
LIN {X 0,Y 409.407,Z 396.033,A -85,B 0,C 180,E1 19965.141,E2 19965.141} C_VEL
LIN {X 0,Y 409.423,Z 396.032,A -85,B 0,C 180,E1 19961.342,E2 19961.342} C_VEL
LIN {X 0,Y 409.391,Z 396.037,A -85,B 0,C 180,E1 19957.604,E2 19957.604} C_VEL
LIN {X 0,Y 409.379,Z 396.043,A -85,B 0,C 180,E1 19953.764,E2 19953.764} C_VEL
LIN {X 0,Y 409.37,Z 395.99,A -85,B 0,C 180,E1 19949.84,E2 19949.84} C_VEL
LIN {X 0,Y 409.413,Z 396.288,A -85,B 0,C 180,E1 19947.667,E2 19947.667} C_VEL
LIN {X 0,Y 410.901,Z 399.768,A -85,B 0,C 180,E1 19946.637,E2 19946.637} C_VEL
LIN {X 0,Y 412.481,Z 401.639,A -85,B 0,C 180,E1 19945.947,E2 19945.947} C_VEL
LIN {X 0,Y 414.314,Z 405.342,A -85,B 0,C 180,E1 19944.945,E2 19944.945} C_VEL
LIN {X 0,Y 415.541,Z 407.181,A -85,B 0,C 180,E1 19944.388,E2 19944.388} C_VEL
LIN {X 0,Y 417.933,Z 411.27,A -85,B 0,C 180,E1 19943.266,E2 19943.266} C_VEL
LIN {X 0,Y 423.663,Z 422.177,A -85,B 0,C 180,E1 19940.591,E2 19940.591} C_VEL
LIN {X 0,Y 428.141,Z 430.907,A -85,B 0,C 180,E1 19938.631,E2 19938.631} C_VEL
LIN {X 0,Y 434.141,Z 443.236,A -85,B 0,C 180,E1 19936.114,E2 19936.114} C_VEL
LIN {X 0,Y 441.066,Z 458.771,A -85,B 0,C 180,E1 19933.307,E2 19933.307} C_VEL
LIN {X 0,Y 443.204,Z 464.206,A -85,B 0,C 180,E1 19932.419,E2 19932.419} C_VEL
LIN {X 0,Y 442.68,Z 469.941,A -85,B 0,C 180,E1 19931.96,E2 19931.96} C_VEL
LIN {X 0,Y 448.067,Z 505.697,A -85,B 0,C 180,E1 19930.454,E2 19930.454} C_VEL
LIN {X 0,Y 443.066,Z 720.925,A -85,B 0,C 180,E1 19926.937,E2 19926.937} C_VEL
LIN {X 0,Y 442.366,Z 748.99,A -85,B 0,C 180,E1 19926.421,E2 19926.421} C_VEL
LIN {X 0,Y 441.26,Z 769.473,A -85,B 0,C 180,E1 19925.816,E2 19925.816} C_VEL
LIN {X 0,Y 440.416,Z 779.867,A -85,B 0,C 180,E1 19925.414,E2 19925.414} C_VEL
LIN {X 0,Y 438.992,Z 787.303,A -85,B 0,C 180,E1 19925.184,E2 19925.184} C_VEL
LIN {X 0,Y 432.241,Z 806.015,A -85,B 0,C 180,E1 19924.722,E2 19924.722} C_VEL
LIN {X 0,Y 430.565,Z 813.008,A -85,B 0,C 180,E1 19924.378,E2 19924.378} C_VEL
LIN {X 0,Y 427.751,Z 830.967,A -85,B 0,C 180,E1 19923.08,E2 19923.08} C_VEL
LIN {X 0,Y 424.527,Z 848.597,A -85,B 0,C 180,E1 19921.525,E2 19921.525} C_VEL
LIN {X 0,Y 421.231,Z 864.62,A -85,B 0,C 180,E1 19919.821,E2 19919.821} C_VEL
LIN {X 0,Y 417.755,Z 880.214,A -85,B 0,C 180,E1 19917.822,E2 19917.822} C_VEL
LIN {X 0,Y 414.476,Z 893.717,A -85,B 0,C 180,E1 19915.736,E2 19915.736} C_VEL
LIN {X 0,Y 411.272,Z 906.665,A -85,B 0,C 180,E1 19913.346,E2 19913.346} C_VEL
LIN {X 0,Y 408.342,Z 918.45,A -85,B 0,C 180,E1 19910.713,E2 19910.713} C_VEL
LIN {X 0,Y 406.018,Z 928.152,A -85,B 0,C 180,E1 19908.077,E2 19908.077} C_VEL
LIN {X 0,Y 404.105,Z 936.693,A -85,B 0,C 180,E1 19905.205,E2 19905.205} C_VEL
LIN {X 0,Y 402.657,Z 943.693,A -85,B 0,C 180,E1 19902.185,E2 19902.185} C_VEL
LIN {X 0,Y 401.753,Z 948.944,A -85,B 0,C 180,E1 19899.165,E2 19899.165} C_VEL
LIN {X 0,Y 401.201,Z 952.756,A -85,B 0,C 180,E1 19896.008,E2 19896.008} C_VEL
LIN {X 0,Y 400.942,Z 954.954,A -85,B 0,C 180,E1 19892.859,E2 19892.859} C_VEL
LIN {X 0,Y 400.879,Z 955.622,A -85,B 0,C 180,E1 19889.714,E2 19889.714} C_VEL
LIN {X 0,Y 400.974,Z 954.768,A -85,B 0,C 180,E1 19886.569,E2 19886.569} C_VEL
LIN {X 0,Y 401.284,Z 952.304,A -85,B 0,C 180,E1 19883.419,E2 19883.419} C_VEL
LIN {X 0,Y 401.836,Z 948.433,A -85,B 0,C 180,E1 19880.403,E2 19880.403} C_VEL
LIN {X 0,Y 402.85,Z 942.665,A -85,B 0,C 180,E1 19877.238,E2 19877.238} C_VEL
LIN {X 0,Y 404.372,Z 935.34,A -85,B 0,C 180,E1 19874.217,E2 19874.217} C_VEL
LIN {X 0,Y 406.3,Z 927.022,A -85,B 0,C 180,E1 19871.491,E2 19871.491} C_VEL
LIN {X 0,Y 408.862,Z 916.502,A -85,B 0,C 180,E1 19868.706,E2 19868.706} C_VEL
LIN {X 0,Y 411.713,Z 905.007,A -85,B 0,C 180,E1 19866.225,E2 19866.225} C_VEL
LIN {X 0,Y 414.764,Z 892.55,A -85,B 0,C 180,E1 19863.976,E2 19863.976} C_VEL
LIN {X 0,Y 418.168,Z 878.431,A -85,B 0,C 180,E1 19861.843,E2 19861.843} C_VEL
LIN {X 0,Y 421.616,Z 863.013,A -85,B 0,C 180,E1 19859.894,E2 19859.894} C_VEL
LIN {X 0,Y 424.938,Z 846.675,A -85,B 0,C 180,E1 19858.193,E2 19858.193} C_VEL
LIN {X 0,Y 428.031,Z 829.429,A -85,B 0,C 180,E1 19856.705,E2 19856.705} C_VEL
LIN {X 0,Y 430.804,Z 811.365,A -85,B 0,C 180,E1 19855.426,E2 19855.426} C_VEL
LIN {X 0,Y 433.236,Z 792.283,A -85,B 0,C 180,E1 19854.348,E2 19854.348} C_VEL
LIN {X 0,Y 435.045,Z 772.881,A -85,B 0,C 180,E1 19853.51,E2 19853.51} C_VEL
LIN {X 0,Y 436.3,Z 752.474,A -85,B 0,C 180,E1 19852.866,E2 19852.866} C_VEL
LIN {X 0,Y 437.049,Z 727.795,A -85,B 0,C 180,E1 19852.373,E2 19852.373} C_VEL
LIN {X 0,Y 442.466,Z 509.233,A -85,B 0,C 180,E1 19848.763,E2 19848.763} C_VEL
LIN {X 0,Y 442.312,Z 504.855,A -85,B 0,C 180,E1 19848.649,E2 19848.649} C_VEL
LIN {X 0,Y 436.976,Z 469.003,A -85,B 0,C 180,E1 19847.072,E2 19847.072} C_VEL
LIN {X 0,Y 436.833,Z 467.495,A -85,B 0,C 180,E1 19846.9,E2 19846.9} C_VEL
LIN {X 0,Y 430.324,Z 452.32,A -85,B 0,C 180,E1 19844.191,E2 19844.191} C_VEL
LIN {X 0,Y 424.056,Z 438.852,A -85,B 0,C 180,E1 19841.495,E2 19841.495} C_VEL
LIN {X 0,Y 417.805,Z 426.323,A -85,B 0,C 180,E1 19838.654,E2 19838.654} C_VEL
LIN {X 0,Y 412.54,Z 416.796,A -85,B 0,C 180,E1 19836.188,E2 19836.188} C_VEL
LIN {X 0,Y 410.111,Z 412.272,A -85,B 0,C 180,E1 19834.956,E2 19834.956} C_VEL
LIN {X 0,Y 407.838,Z 408.314,A -85,B 0,C 180,E1 19833.788,E2 19833.788} C_VEL
LIN {X 0,Y 405.109,Z 404.015,A -85,B 0,C 180,E1 19832.384,E2 19832.384} C_VEL
LIN {X 0,Y 404.148,Z 402.059,A -85,B 0,C 180,E1 19831.801,E2 19831.801} C_VEL
LIN {X 0,Y 401.871,Z 398.733,A -85,B 0,C 180,E1 19830.587,E2 19830.587} C_VEL
LIN {X 0,Y 401.457,Z 397.105,A -85,B 0,C 180,E1 19829.995,E2 19829.995} C_VEL
LIN {X 0,Y 401.444,Z 397.029,A -85,B 0,C 180,E1 19825.999,E2 19825.999} C_VEL
LIN {X 0,Y 401.445,Z 397.025,A -85,B 0,C 180,E1 19822.092,E2 19822.092} C_VEL
LIN {X 0,Y 401.464,Z 397.023,A -85,B 0,C 180,E1 19818.289,E2 19818.289} C_VEL
LIN {X 0,Y 401.492,Z 397.02,A -85,B 0,C 180,E1 19814.421,E2 19814.421} C_VEL
LIN {X 0,Y 401.482,Z 397.021,A -85,B 0,C 180,E1 19810.475,E2 19810.475} C_VEL
LIN {X 0,Y 401.452,Z 397.025,A -85,B 0,C 180,E1 19806.723,E2 19806.723} C_VEL
LIN {X 0,Y 401.438,Z 397.028,A -85,B 0,C 180,E1 19802.836,E2 19802.836} C_VEL
LIN {X 0,Y 401.436,Z 397.029,A -85,B 0,C 180,E1 19799.001,E2 19799.001} C_VEL
LIN {X 0,Y 401.447,Z 397.029,A -85,B 0,C 180,E1 19795.143,E2 19795.143} C_VEL
LIN {X 0,Y 401.479,Z 397.025,A -85,B 0,C 180,E1 19791.383,E2 19791.383} C_VEL
LIN {X 0,Y 401.475,Z 396.964,A -85,B 0,C 180,E1 19787.341,E2 19787.341} C_VEL
LIN {X 0,Y 401.464,Z 397.039,A -85,B 0,C 180,E1 19783.506,E2 19783.506} C_VEL
LIN {X 0,Y 401.435,Z 397.007,A -85,B 0,C 180,E1 19779.745,E2 19779.745} C_VEL
LIN {X 0,Y 401.578,Z 397.613,A -85,B 0,C 180,E1 19779.143,E2 19779.143} C_VEL
LIN {X 0,Y 403.112,Z 401.009,A -85,B 0,C 180,E1 19778.158,E2 19778.158} C_VEL
LIN {X 0,Y 405.06,Z 402.92,A -85,B 0,C 180,E1 19777.352,E2 19777.352} C_VEL
LIN {X 0,Y 406.838,Z 406.623,A -85,B 0,C 180,E1 19776.385,E2 19776.385} C_VEL
LIN {X 0,Y 408.53,Z 408.406,A -85,B 0,C 180,E1 19775.722,E2 19775.722} C_VEL
LIN {X 0,Y 410.807,Z 412.605,A -85,B 0,C 180,E1 19774.637,E2 19774.637} C_VEL
LIN {X 0,Y 412.101,Z 414.49,A -85,B 0,C 180,E1 19774.105,E2 19774.105} C_VEL
LIN {X 0,Y 415.264,Z 419.762,A -85,B 0,C 180,E1 19772.776,E2 19772.776} C_VEL
LIN {X 0,Y 418.882,Z 425.921,A -85,B 0,C 180,E1 19771.329,E2 19771.329} C_VEL
LIN {X 0,Y 423.414,Z 433.476,A -85,B 0,C 180,E1 19769.646,E2 19769.646} C_VEL
LIN {X 0,Y 432.063,Z 449.283,A -85,B 0,C 180,E1 19766.581,E2 19766.581} C_VEL
LIN {X 0,Y 440.375,Z 465.801,A -85,B 0,C 180,E1 19763.821,E2 19763.821} C_VEL
LIN {X 0,Y 446.612,Z 476.095,A -85,B 0,C 180,E1 19762.654,E2 19762.654} C_VEL
LIN {X 0,Y 448.95,Z 504.125,A -85,B 0,C 180,E1 19761.665,E2 19761.665} C_VEL
LIN {X 0,Y 441.598,Z 694.777,A -85,B 0,C 180,E1 19757.998,E2 19757.998} C_VEL
LIN {X 0,Y 437.294,Z 806.365,A -85,B 0,C 180,E1 19755.811,E2 19755.811} C_VEL
LIN {X 0,Y 435.368,Z 829.976,A -85,B 0,C 180,E1 19755.152,E2 19755.152} C_VEL
LIN {X 0,Y 433.018,Z 852.673,A -85,B 0,C 180,E1 19754.306,E2 19754.306} C_VEL
LIN {X 0,Y 430.351,Z 874.336,A -85,B 0,C 180,E1 19753.267,E2 19753.267} C_VEL
LIN {X 0,Y 427.243,Z 897.194,A -85,B 0,C 180,E1 19751.91,E2 19751.91} C_VEL
LIN {X 0,Y 424.012,Z 919.229,A -85,B 0,C 180,E1 19750.338,E2 19750.338} C_VEL
LIN {X 0,Y 420.636,Z 940.494,A -85,B 0,C 180,E1 19748.52,E2 19748.52} C_VEL
LIN {X 0,Y 417.164,Z 962.084,A -85,B 0,C 180,E1 19746.359,E2 19746.359} C_VEL
LIN {X 0,Y 413.93,Z 982.043,A -85,B 0,C 180,E1 19744.054,E2 19744.054} C_VEL
LIN {X 0,Y 411.063,Z 1000.213,A -85,B 0,C 180,E1 19741.644,E2 19741.644} C_VEL
LIN {X 0,Y 408.376,Z 1017.443,A -85,B 0,C 180,E1 19738.998,E2 19738.998} C_VEL
LIN {X 0,Y 406.346,Z 1030.953,A -85,B 0,C 180,E1 19736.605,E2 19736.605} C_VEL
LIN {X 0,Y 404.387,Z 1044.641,A -85,B 0,C 180,E1 19733.767,E2 19733.767} C_VEL
LIN {X 0,Y 402.936,Z 1055.778,A -85,B 0,C 180,E1 19731.089,E2 19731.089} C_VEL
LIN {X 0,Y 401.718,Z 1066.37,A -85,B 0,C 180,E1 19728.053,E2 19728.053} C_VEL
LIN {X 0,Y 400.929,Z 1074.311,A -85,B 0,C 180,E1 19725.328,E2 19725.328} C_VEL
LIN {X 0,Y 400.357,Z 1081.89,A -85,B 0,C 180,E1 19722.11,E2 19722.11} C_VEL
LIN {X 0,Y 400.067,Z 1086.91,A -85,B 0,C 180,E1 19719.349,E2 19719.349} C_VEL
LIN {X 0,Y 399.948,Z 1090.78,A -85,B 0,C 180,E1 19716.459,E2 19716.459} C_VEL
LIN {X 0,Y 399.89,Z 1093.037,A -85,B 0,C 180,E1 19713.44,E2 19713.44} C_VEL
LIN {X 0,Y 399.889,Z 1093.87,A -85,B 0,C 180,E1 19710.86,E2 19710.86} C_VEL
LIN {X 0,Y 399.91,Z 1093.592,A -85,B 0,C 180,E1 19707.707,E2 19707.707} C_VEL
LIN {X 0,Y 399.919,Z 1091.895,A -85,B 0,C 180,E1 19704.836,E2 19704.836} C_VEL
LIN {X 0,Y 399.976,Z 1089.202,A -85,B 0,C 180,E1 19702.242,E2 19702.242} C_VEL
LIN {X 0,Y 400.195,Z 1084.49,A -85,B 0,C 180,E1 19699.2,E2 19699.2} C_VEL
LIN {X 0,Y 400.606,Z 1078.334,A -85,B 0,C 180,E1 19696.284,E2 19696.284} C_VEL
LIN {X 0,Y 401.305,Z 1070.276,A -85,B 0,C 180,E1 19693.201,E2 19693.201} C_VEL
LIN {X 0,Y 402.327,Z 1060.67,A -85,B 0,C 180,E1 19690.246,E2 19690.246} C_VEL
LIN {X 0,Y 403.683,Z 1049.883,A -85,B 0,C 180,E1 19687.424,E2 19687.424} C_VEL
LIN {X 0,Y 405.473,Z 1036.983,A -85,B 0,C 180,E1 19684.591,E2 19684.591} C_VEL
LIN {X 0,Y 407.582,Z 1022.807,A -85,B 0,C 180,E1 19681.9,E2 19681.9} C_VEL
LIN {X 0,Y 410.003,Z 1007.066,A -85,B 0,C 180,E1 19679.357,E2 19679.357} C_VEL
LIN {X 0,Y 412.853,Z 988.854,A -85,B 0,C 180,E1 19676.815,E2 19676.815} C_VEL
LIN {X 0,Y 416.194,Z 967.989,A -85,B 0,C 180,E1 19674.283,E2 19674.283} C_VEL
LIN {X 0,Y 419.403,Z 948.245,A -85,B 0,C 180,E1 19672.215,E2 19672.215} C_VEL
LIN {X 0,Y 422.864,Z 926.274,A -85,B 0,C 180,E1 19670.238,E2 19670.238} C_VEL
LIN {X 0,Y 426.208,Z 904.549,A -85,B 0,C 180,E1 19668.581,E2 19668.581} C_VEL
LIN {X 0,Y 429.042,Z 884.383,A -85,B 0,C 180,E1 19667.3,E2 19667.3} C_VEL
LIN {X 0,Y 431.939,Z 861.853,A -85,B 0,C 180,E1 19666.109,E2 19666.109} C_VEL
LIN {X 0,Y 434.41,Z 839.443,A -85,B 0,C 180,E1 19665.171,E2 19665.171} C_VEL
LIN {X 0,Y 436.611,Z 815.4,A -85,B 0,C 180,E1 19664.421,E2 19664.421} C_VEL
LIN {X 0,Y 438.015,Z 790.861,A -85,B 0,C 180,E1 19663.861,E2 19663.861} C_VEL
LIN {X 0,Y 445.934,Z 581.799,A -85,B 0,C 180,E1 19659.82,E2 19659.82} C_VEL
LIN {X 0,Y 448.849,Z 501.532,A -85,B 0,C 180,E1 19658.269,E2 19658.269} C_VEL
LIN {X 0,Y 446.403,Z 475.488,A -85,B 0,C 180,E1 19657.311,E2 19657.311} C_VEL
LIN {X 0,Y 440.353,Z 465.788,A -85,B 0,C 180,E1 19656.181,E2 19656.181} C_VEL
LIN {X 0,Y 432.018,Z 449.242,A -85,B 0,C 180,E1 19653.423,E2 19653.423} C_VEL
LIN {X 0,Y 424.739,Z 436.025,A -85,B 0,C 180,E1 19650.876,E2 19650.876} C_VEL
LIN {X 0,Y 419.845,Z 427.505,A -85,B 0,C 180,E1 19649.066,E2 19649.066} C_VEL
LIN {X 0,Y 416.812,Z 422.454,A -85,B 0,C 180,E1 19647.889,E2 19647.889} C_VEL
LIN {X 0,Y 413.884,Z 417.565,A -85,B 0,C 180,E1 19646.701,E2 19646.701} C_VEL
LIN {X 0,Y 411.078,Z 412.926,A -85,B 0,C 180,E1 19645.5,E2 19645.5} C_VEL
LIN {X 0,Y 408.7,Z 408.91,A -85,B 0,C 180,E1 19644.421,E2 19644.421} C_VEL
LIN {X 0,Y 405.649,Z 404.611,A -85,B 0,C 180,E1 19643.073,E2 19643.073} C_VEL
LIN {X 0,Y 405.005,Z 402.773,A -85,B 0,C 180,E1 19642.651,E2 19642.651} C_VEL
LIN {X 0,Y 402.486,Z 400.079,A -85,B 0,C 180,E1 19641.571,E2 19641.571} C_VEL
LIN {X 0,Y 401.517,Z 397.333,A -85,B 0,C 180,E1 19640.784,E2 19640.784} C_VEL
LIN {X 0,Y 401.455,Z 396.979,A -85,B 0,C 180,E1 19638.59,E2 19638.59} C_VEL
LIN {X 0,Y 401.488,Z 396.982,A -85,B 0,C 180,E1 19634.715,E2 19634.715} C_VEL
LIN {X 0,Y 401.473,Z 397.004,A -85,B 0,C 180,E1 19630.62,E2 19630.62} C_VEL
LIN {X 0,Y 401.458,Z 397.025,A -85,B 0,C 180,E1 19626.722,E2 19626.722} C_VEL
LIN {X 0,Y 401.44,Z 397.034,A -85,B 0,C 180,E1 19622.84,E2 19622.84} C_VEL
LIN {X 0,Y 401.433,Z 397.038,A -85,B 0,C 180,E1 19619.001,E2 19619.001} C_VEL
LIN {X 0,Y 401.435,Z 397.041,A -85,B 0,C 180,E1 19614.998,E2 19614.998} C_VEL
LIN {X 0,Y 401.456,Z 397.035,A -85,B 0,C 180,E1 19611.261,E2 19611.261} C_VEL
LIN {X 0,Y 401.477,Z 397.035,A -85,B 0,C 180,E1 19607.34,E2 19607.34} C_VEL
LIN {X 0,Y 401.481,Z 397.037,A -85,B 0,C 180,E1 19603.5,E2 19603.5} C_VEL
LIN {X 0,Y 401.463,Z 397.042,A -85,B 0,C 180,E1 19599.593,E2 19599.593} C_VEL
LIN {X 0,Y 401.439,Z 397.041,A -85,B 0,C 180,E1 19595.891,E2 19595.891} C_VEL
LIN {X 0,Y 401.44,Z 397.011,A -85,B 0,C 180,E1 19591.917,E2 19591.917} C_VEL
LIN {X 0,Y 401.468,Z 397.237,A -85,B 0,C 180,E1 19589.793,E2 19589.793} C_VEL
LIN {X 0,Y 402.235,Z 399.538,A -85,B 0,C 180,E1 19589.032,E2 19589.032} C_VEL
LIN {X 0,Y 404.752,Z 402.972,A -85,B 0,C 180,E1 19587.752,E2 19587.752} C_VEL
LIN {X 0,Y 406.48,Z 406.419,A -85,B 0,C 180,E1 19586.733,E2 19586.733} C_VEL
LIN {X 0,Y 407.71,Z 407.966,A -85,B 0,C 180,E1 19586.172,E2 19586.172} C_VEL
LIN {X 0,Y 409.87,Z 412,A -85,B 0,C 180,E1 19585.021,E2 19585.021} C_VEL
LIN {X 0,Y 413.677,Z 418.898,A -85,B 0,C 180,E1 19583.134,E2 19583.134} C_VEL
LIN {X 0,Y 418.281,Z 427.444,A -85,B 0,C 180,E1 19580.976,E2 19580.976} C_VEL
LIN {X 0,Y 424.507,Z 439.756,A -85,B 0,C 180,E1 19578.197,E2 19578.197} C_VEL
LIN {X 0,Y 431.72,Z 455.349,A -85,B 0,C 180,E1 19575.129,E2 19575.129} C_VEL
LIN {X 0,Y 437.01,Z 468.203,A -85,B 0,C 180,E1 19572.896,E2 19572.896} C_VEL
LIN {X 0,Y 437.436,Z 472.774,A -85,B 0,C 180,E1 19572.656,E2 19572.656} C_VEL
LIN {X 0,Y 442.491,Z 507.342,A -85,B 0,C 180,E1 19571.174,E2 19571.174} C_VEL
LIN {X 0,Y 437.1,Z 724.074,A -85,B 0,C 180,E1 19567.593,E2 19567.593} C_VEL
LIN {X 0,Y 436.356,Z 750.677,A -85,B 0,C 180,E1 19567.086,E2 19567.086} C_VEL
LIN {X 0,Y 435.186,Z 770.928,A -85,B 0,C 180,E1 19566.472,E2 19566.472} C_VEL
LIN {X 0,Y 433.429,Z 789.973,A -85,B 0,C 180,E1 19565.666,E2 19565.666} C_VEL
LIN {X 0,Y 431.104,Z 808.963,A -85,B 0,C 180,E1 19564.627,E2 19564.627} C_VEL
LIN {X 0,Y 430.565,Z 813.008,A -85,B 0,C 180,E1 19564.378,E2 19564.378} C_VEL
LIN {X 0,Y 428.816,Z 820.033,A -85,B 0,C 180,E1 19564.002,E2 19564.002} C_VEL
LIN {X 0,Y 421.168,Z 837.687,A -85,B 0,C 180,E1 19563.174,E2 19563.174} C_VEL
LIN {X 0,Y 419.178,Z 844.169,A -85,B 0,C 180,E1 19562.687,E2 19562.687} C_VEL
LIN {X 0,Y 415.816,Z 860.273,A -85,B 0,C 180,E1 19561.05,E2 19561.05} C_VEL
LIN {X 0,Y 412.167,Z 876.224,A -85,B 0,C 180,E1 19559.104,E2 19559.104} C_VEL
LIN {X 0,Y 408.737,Z 890.215,A -85,B 0,C 180,E1 19557.065,E2 19557.065} C_VEL
LIN {X 0,Y 405.207,Z 903.966,A -85,B 0,C 180,E1 19554.646,E2 19554.646} C_VEL
LIN {X 0,Y 402.143,Z 915.444,A -85,B 0,C 180,E1 19552.205,E2 19552.205} C_VEL
LIN {X 0,Y 399.378,Z 926.143,A -85,B 0,C 180,E1 19549.449,E2 19549.449} C_VEL
LIN {X 0,Y 397.086,Z 935.33,A -85,B 0,C 180,E1 19546.531,E2 19546.531} C_VEL
LIN {X 0,Y 395.442,Z 942.667,A -85,B 0,C 180,E1 19543.6,E2 19543.6} C_VEL
LIN {X 0,Y 394.26,Z 948.592,A -85,B 0,C 180,E1 19540.521,E2 19540.521} C_VEL
LIN {X 0,Y 393.542,Z 952.975,A -85,B 0,C 180,E1 19537.298,E2 19537.298} C_VEL
LIN {X 0,Y 393.154,Z 955.615,A -85,B 0,C 180,E1 19534.23,E2 19534.23} C_VEL
LIN {X 0,Y 393.007,Z 956.88,A -85,B 0,C 180,E1 19531.004,E2 19531.004} C_VEL
LIN {X 0,Y 393.039,Z 956.644,A -85,B 0,C 180,E1 19527.813,E2 19527.813} C_VEL
LIN {X 0,Y 393.266,Z 954.902,A -85,B 0,C 180,E1 19524.602,E2 19524.602} C_VEL
LIN {X 0,Y 393.775,Z 951.51,A -85,B 0,C 180,E1 19521.384,E2 19521.384} C_VEL
LIN {X 0,Y 394.608,Z 946.672,A -85,B 0,C 180,E1 19518.305,E2 19518.305} C_VEL
LIN {X 0,Y 396.006,Z 940.14,A -85,B 0,C 180,E1 19515.226,E2 19515.226} C_VEL
LIN {X 0,Y 397.968,Z 931.724,A -85,B 0,C 180,E1 19512.151,E2 19512.151} C_VEL
LIN {X 0,Y 400.394,Z 922.262,A -85,B 0,C 180,E1 19509.384,E2 19509.384} C_VEL
LIN {X 0,Y 403.25,Z 911.413,A -85,B 0,C 180,E1 19506.781,E2 19506.781} C_VEL
LIN {X 0,Y 406.472,Z 899.049,A -85,B 0,C 180,E1 19504.346,E2 19504.346} C_VEL
LIN {X 0,Y 409.97,Z 885.242,A -85,B 0,C 180,E1 19502.078,E2 19502.078} C_VEL
LIN {X 0,Y 413.691,Z 869.853,A -85,B 0,C 180,E1 19499.98,E2 19499.98} C_VEL
LIN {X 0,Y 417.063,Z 854.728,A -85,B 0,C 180,E1 19498.249,E2 19498.249} C_VEL
LIN {X 0,Y 420.375,Z 838.027,A -85,B 0,C 180,E1 19496.672,E2 19496.672} C_VEL
LIN {X 0,Y 423.382,Z 820.548,A -85,B 0,C 180,E1 19495.309,E2 19495.309} C_VEL
LIN {X 0,Y 426.015,Z 802.409,A -85,B 0,C 180,E1 19494.156,E2 19494.156} C_VEL
LIN {X 0,Y 428.271,Z 782.731,A -85,B 0,C 180,E1 19493.171,E2 19493.171} C_VEL
LIN {X 0,Y 429.871,Z 762.866,A -85,B 0,C 180,E1 19492.438,E2 19492.438} C_VEL
LIN {X 0,Y 430.841,Z 742.162,A -85,B 0,C 180,E1 19491.906,E2 19491.906} C_VEL
LIN {X 0,Y 437.021,Z 507.828,A -85,B 0,C 180,E1 19487.966,E2 19487.966} C_VEL
LIN {X 0,Y 431.704,Z 472.308,A -85,B 0,C 180,E1 19486.367,E2 19486.367} C_VEL
LIN {X 0,Y 429.347,Z 468.181,A -85,B 0,C 180,E1 19485.83,E2 19485.83} C_VEL
LIN {X 0,Y 422.693,Z 452.768,A -85,B 0,C 180,E1 19482.942,E2 19482.942} C_VEL
LIN {X 0,Y 416.251,Z 439.373,A -85,B 0,C 180,E1 19480.073,E2 19480.073} C_VEL
LIN {X 0,Y 410.499,Z 428.066,A -85,B 0,C 180,E1 19477.337,E2 19477.337} C_VEL
LIN {X 0,Y 407.555,Z 422.766,A -85,B 0,C 180,E1 19475.898,E2 19475.898} C_VEL
LIN {X 0,Y 405.022,Z 418.14,A -85,B 0,C 180,E1 19474.597,E2 19474.597} C_VEL
LIN {X 0,Y 402.299,Z 413.348,A -85,B 0,C 180,E1 19473.147,E2 19473.147} C_VEL
LIN {X 0,Y 400.221,Z 409.707,A -85,B 0,C 180,E1 19471.981,E2 19471.981} C_VEL
LIN {X 0,Y 399.148,Z 408.061,A -85,B 0,C 180,E1 19471.402,E2 19471.402} C_VEL
LIN {X 0,Y 397.152,Z 404.709,A -85,B 0,C 180,E1 19470.233,E2 19470.233} C_VEL
LIN {X 0,Y 396.218,Z 403.032,A -85,B 0,C 180,E1 19469.644,E2 19469.644} C_VEL
LIN {X 0,Y 393.888,Z 399.636,A -85,B 0,C 180,E1 19468.256,E2 19468.256} C_VEL
LIN {X 0,Y 393.53,Z 398.091,A -85,B 0,C 180,E1 19467.595,E2 19467.595} C_VEL
LIN {X 0,Y 393.511,Z 398.032,A -85,B 0,C 180,E1 19463.67,E2 19463.67} C_VEL
LIN {X 0,Y 393.504,Z 398.025,A -85,B 0,C 180,E1 19459.752,E2 19459.752} C_VEL
LIN {X 0,Y 393.504,Z 398.019,A -85,B 0,C 180,E1 19455.776,E2 19455.776} C_VEL
LIN {X 0,Y 393.521,Z 398.014,A -85,B 0,C 180,E1 19451.981,E2 19451.981} C_VEL
LIN {X 0,Y 393.539,Z 398.011,A -85,B 0,C 180,E1 19448.033,E2 19448.033} C_VEL
LIN {X 0,Y 393.542,Z 398.01,A -85,B 0,C 180,E1 19444.08,E2 19444.08} C_VEL
LIN {X 0,Y 393.55,Z 398.007,A -85,B 0,C 180,E1 19440,E2 19440} C_VEL
LIN {X 0,Y 393.522,Z 398.011,A -85,B 0,C 180,E1 19436.067,E2 19436.067} C_VEL
LIN {X 0,Y 393.501,Z 398.013,A -85,B 0,C 180,E1 19432.261,E2 19432.261} C_VEL
LIN {X 0,Y 393.489,Z 397.971,A -85,B 0,C 180,E1 19428.42,E2 19428.42} C_VEL
LIN {X 0,Y 393.493,Z 398.003,A -85,B 0,C 180,E1 19424.374,E2 19424.374} C_VEL
LIN {X 0,Y 393.521,Z 398.16,A -85,B 0,C 180,E1 19421.789,E2 19421.789} C_VEL
LIN {X 0,Y 393.921,Z 399.622,A -85,B 0,C 180,E1 19421.195,E2 19421.195} C_VEL
LIN {X 0,Y 395.873,Z 402.735,A -85,B 0,C 180,E1 19420.065,E2 19420.065} C_VEL
LIN {X 0,Y 397.34,Z 404.28,A -85,B 0,C 180,E1 19419.373,E2 19419.373} C_VEL
LIN {X 0,Y 399.275,Z 408.044,A -85,B 0,C 180,E1 19418.247,E2 19418.247} C_VEL
LIN {X 0,Y 400.85,Z 409.739,A -85,B 0,C 180,E1 19417.566,E2 19417.566} C_VEL
LIN {X 0,Y 402.985,Z 413.686,A -85,B 0,C 180,E1 19416.456,E2 19416.456} C_VEL
LIN {X 0,Y 404.467,Z 415.702,A -85,B 0,C 180,E1 19415.81,E2 19415.81} C_VEL
LIN {X 0,Y 407.832,Z 421.285,A -85,B 0,C 180,E1 19414.283,E2 19414.283} C_VEL
LIN {X 0,Y 411.064,Z 426.733,A -85,B 0,C 180,E1 19412.905,E2 19412.905} C_VEL
LIN {X 0,Y 414.248,Z 432.119,A -85,B 0,C 180,E1 19411.609,E2 19411.609} C_VEL
LIN {X 0,Y 418.72,Z 439.713,A -85,B 0,C 180,E1 19409.904,E2 19409.904} C_VEL
LIN {X 0,Y 426.873,Z 454.823,A -85,B 0,C 180,E1 19406.925,E2 19406.925} C_VEL
LIN {X 0,Y 433.285,Z 467.309,A -85,B 0,C 180,E1 19404.808,E2 19404.808} C_VEL
LIN {X 0,Y 441.368,Z 480.291,A -85,B 0,C 180,E1 19403.285,E2 19403.285} C_VEL
LIN {X 0,Y 443.364,Z 505.507,A -85,B 0,C 180,E1 19402.385,E2 19402.385} C_VEL
LIN {X 0,Y 435.662,Z 696.019,A -85,B 0,C 180,E1 19398.685,E2 19398.685} C_VEL
LIN {X 0,Y 431.229,Z 805.419,A -85,B 0,C 180,E1 19396.517,E2 19396.517} C_VEL
LIN {X 0,Y 429.248,Z 828.908,A -85,B 0,C 180,E1 19395.856,E2 19395.856} C_VEL
LIN {X 0,Y 426.844,Z 851.174,A -85,B 0,C 180,E1 19395.026,E2 19395.026} C_VEL
LIN {X 0,Y 423.96,Z 873.463,A -85,B 0,C 180,E1 19393.949,E2 19393.949} C_VEL
LIN {X 0,Y 420.595,Z 896.752,A -85,B 0,C 180,E1 19392.548,E2 19392.548} C_VEL
LIN {X 0,Y 417.203,Z 918.664,A -85,B 0,C 180,E1 19390.955,E2 19390.955} C_VEL
LIN {X 0,Y 413.788,Z 938.987,A -85,B 0,C 180,E1 19389.189,E2 19389.189} C_VEL
LIN {X 0,Y 410.12,Z 960.295,A -85,B 0,C 180,E1 19387.026,E2 19387.026} C_VEL
LIN {X 0,Y 406.745,Z 979.836,A -85,B 0,C 180,E1 19384.725,E2 19384.725} C_VEL
LIN {X 0,Y 403.579,Z 998.329,A -85,B 0,C 180,E1 19382.186,E2 19382.186} C_VEL
LIN {X 0,Y 400.714,Z 1015.885,A -85,B 0,C 180,E1 19379.443,E2 19379.443} C_VEL
LIN {X 0,Y 398.613,Z 1029.486,A -85,B 0,C 180,E1 19377.002,E2 19377.002} C_VEL
LIN {X 0,Y 396.572,Z 1043.33,A -85,B 0,C 180,E1 19374.107,E2 19374.107} C_VEL
LIN {X 0,Y 394.993,Z 1055.097,A -85,B 0,C 180,E1 19371.222,E2 19371.222} C_VEL
LIN {X 0,Y 393.786,Z 1065.372,A -85,B 0,C 180,E1 19368.199,E2 19368.199} C_VEL
LIN {X 0,Y 392.93,Z 1073.931,A -85,B 0,C 180,E1 19365.195,E2 19365.195} C_VEL
LIN {X 0,Y 392.413,Z 1080.971,A -85,B 0,C 180,E1 19362.06,E2 19362.06} C_VEL
LIN {X 0,Y 392.143,Z 1085.927,A -85,B 0,C 180,E1 19359.244,E2 19359.244} C_VEL
LIN {X 0,Y 392.016,Z 1089.983,A -85,B 0,C 180,E1 19356.003,E2 19356.003} C_VEL
LIN {X 0,Y 391.964,Z 1091.976,A -85,B 0,C 180,E1 19353.364,E2 19353.364} C_VEL
LIN {X 0,Y 391.952,Z 1092.865,A -85,B 0,C 180,E1 19350.731,E2 19350.731} C_VEL
LIN {X 0,Y 391.978,Z 1092.518,A -85,B 0,C 180,E1 19347.661,E2 19347.661} C_VEL
LIN {X 0,Y 392.005,Z 1090.64,A -85,B 0,C 180,E1 19344.731,E2 19344.731} C_VEL
LIN {X 0,Y 392.098,Z 1087.61,A -85,B 0,C 180,E1 19341.938,E2 19341.938} C_VEL
LIN {X 0,Y 392.312,Z 1082.431,A -85,B 0,C 180,E1 19338.682,E2 19338.682} C_VEL
LIN {X 0,Y 392.725,Z 1076.439,A -85,B 0,C 180,E1 19335.853,E2 19335.853} C_VEL
LIN {X 0,Y 393.472,Z 1068.161,A -85,B 0,C 180,E1 19332.704,E2 19332.704} C_VEL
LIN {X 0,Y 394.502,Z 1058.887,A -85,B 0,C 180,E1 19329.837,E2 19329.837} C_VEL
LIN {X 0,Y 396.014,Z 1047.211,A -85,B 0,C 180,E1 19326.783,E2 19326.783} C_VEL
LIN {X 0,Y 397.794,Z 1034.851,A -85,B 0,C 180,E1 19324.065,E2 19324.065} C_VEL
LIN {X 0,Y 400.166,Z 1019.504,A -85,B 0,C 180,E1 19321.168,E2 19321.168} C_VEL
LIN {X 0,Y 402.744,Z 1003.489,A -85,B 0,C 180,E1 19318.577,E2 19318.577} C_VEL
LIN {X 0,Y 405.863,Z 984.938,A -85,B 0,C 180,E1 19315.951,E2 19315.951} C_VEL
LIN {X 0,Y 409.196,Z 965.687,A -85,B 0,C 180,E1 19313.575,E2 19313.575} C_VEL
LIN {X 0,Y 412.522,Z 946.422,A -85,B 0,C 180,E1 19311.524,E2 19311.524} C_VEL
LIN {X 0,Y 415.974,Z 925.777,A -85,B 0,C 180,E1 19309.636,E2 19309.636} C_VEL
LIN {X 0,Y 419.517,Z 904.138,A -85,B 0,C 180,E1 19307.954,E2 19307.954} C_VEL
LIN {X 0,Y 422.591,Z 883.324,A -85,B 0,C 180,E1 19306.613,E2 19306.613} C_VEL
LIN {X 0,Y 425.689,Z 860.306,A -85,B 0,C 180,E1 19305.388,E2 19305.388} C_VEL
LIN {X 0,Y 428.32,Z 837.667,A -85,B 0,C 180,E1 19304.44,E2 19304.44} C_VEL
LIN {X 0,Y 430.559,Z 814.046,A -85,B 0,C 180,E1 19303.708,E2 19303.708} C_VEL
LIN {X 0,Y 432.022,Z 788.791,A -85,B 0,C 180,E1 19303.131,E2 19303.131} C_VEL
LIN {X 0,Y 440.294,Z 580.775,A -85,B 0,C 180,E1 19299.068,E2 19299.068} C_VEL
LIN {X 0,Y 443.259,Z 502.901,A -85,B 0,C 180,E1 19297.547,E2 19297.547} C_VEL
LIN {X 0,Y 441.122,Z 479.614,A -85,B 0,C 180,E1 19296.673,E2 19296.673} C_VEL
LIN {X 0,Y 432.379,Z 465.886,A -85,B 0,C 180,E1 19294.993,E2 19294.993} C_VEL
LIN {X 0,Y 425.011,Z 451.316,A -85,B 0,C 180,E1 19292.437,E2 19292.437} C_VEL
LIN {X 0,Y 417.624,Z 437.85,A -85,B 0,C 180,E1 19289.708,E2 19289.708} C_VEL
LIN {X 0,Y 412.203,Z 428.661,A -85,B 0,C 180,E1 19287.6,E2 19287.6} C_VEL
LIN {X 0,Y 409.315,Z 423.786,A -85,B 0,C 180,E1 19286.396,E2 19286.396} C_VEL
LIN {X 0,Y 406.514,Z 419.192,A -85,B 0,C 180,E1 19285.182,E2 19285.182} C_VEL
LIN {X 0,Y 403.56,Z 414.323,A -85,B 0,C 180,E1 19283.818,E2 19283.818} C_VEL
LIN {X 0,Y 401.215,Z 410.795,A -85,B 0,C 180,E1 19282.722,E2 19282.722} C_VEL
LIN {X 0,Y 400.48,Z 409.237,A -85,B 0,C 180,E1 19282.302,E2 19282.302} C_VEL
LIN {X 0,Y 398.106,Z 406.285,A -85,B 0,C 180,E1 19281.202,E2 19281.202} C_VEL
LIN {X 0,Y 397.02,Z 403.714,A -85,B 0,C 180,E1 19280.49,E2 19280.49} C_VEL
LIN {X 0,Y 394.464,Z 400.867,A -85,B 0,C 180,E1 19279.239,E2 19279.239} C_VEL
LIN {X 0,Y 393.544,Z 398.271,A -85,B 0,C 180,E1 19278.363,E2 19278.363} C_VEL
LIN {X 0,Y 393.532,Z 397.966,A -85,B 0,C 180,E1 19274.568,E2 19274.568} C_VEL
LIN {X 0,Y 393.535,Z 397.994,A -85,B 0,C 180,E1 19270.497,E2 19270.497} C_VEL
LIN {X 0,Y 393.534,Z 398.014,A -85,B 0,C 180,E1 19266.565,E2 19266.565} C_VEL
LIN {X 0,Y 393.514,Z 398.024,A -85,B 0,C 180,E1 19262.621,E2 19262.621} C_VEL
LIN {X 0,Y 393.497,Z 398.029,A -85,B 0,C 180,E1 19258.835,E2 19258.835} C_VEL
LIN {X 0,Y 393.496,Z 398.031,A -85,B 0,C 180,E1 19254.897,E2 19254.897} C_VEL
LIN {X 0,Y 393.502,Z 398.033,A -85,B 0,C 180,E1 19250.936,E2 19250.936} C_VEL
LIN {X 0,Y 393.517,Z 398.032,A -85,B 0,C 180,E1 19247.079,E2 19247.079} C_VEL
LIN {X 0,Y 393.548,Z 398.028,A -85,B 0,C 180,E1 19243.301,E2 19243.301} C_VEL
LIN {X 0,Y 393.553,Z 398.019,A -85,B 0,C 180,E1 19239.164,E2 19239.164} C_VEL
LIN {X 0,Y 393.534,Z 398.015,A -85,B 0,C 180,E1 19235.214,E2 19235.214} C_VEL
LIN {X 0,Y 393.537,Z 398.266,A -85,B 0,C 180,E1 19232.087,E2 19232.087} C_VEL
LIN {X 0,Y 395.148,Z 401.857,A -85,B 0,C 180,E1 19230.767,E2 19230.767} C_VEL
LIN {X 0,Y 397.001,Z 404.263,A -85,B 0,C 180,E1 19229.753,E2 19229.753} C_VEL
LIN {X 0,Y 399.202,Z 408.14,A -85,B 0,C 180,E1 19228.434,E2 19228.434} C_VEL
LIN {X 0,Y 400.255,Z 409.834,A -85,B 0,C 180,E1 19227.853,E2 19227.853} C_VEL
LIN {X 0,Y 402.722,Z 413.837,A -85,B 0,C 180,E1 19226.534,E2 19226.534} C_VEL
LIN {X 0,Y 405.098,Z 418.251,A -85,B 0,C 180,E1 19225.239,E2 19225.239} C_VEL
LIN {X 0,Y 409.053,Z 425.625,A -85,B 0,C 180,E1 19223.211,E2 19223.211} C_VEL
LIN {X 0,Y 413.315,Z 433.633,A -85,B 0,C 180,E1 19221.166,E2 19221.166} C_VEL
LIN {X 0,Y 419.237,Z 445.44,A -85,B 0,C 180,E1 19218.469,E2 19218.469} C_VEL
LIN {X 0,Y 426.134,Z 460.57,A -85,B 0,C 180,E1 19215.447,E2 19215.447} C_VEL
LIN {X 0,Y 430.159,Z 469.833,A -85,B 0,C 180,E1 19213.827,E2 19213.827} C_VEL
LIN {X 0,Y 431.873,Z 472.982,A -85,B 0,C 180,E1 19213.488,E2 19213.488} C_VEL
LIN {X 0,Y 436.994,Z 508.784,A -85,B 0,C 180,E1 19211.916,E2 19211.916} C_VEL
LIN {X 0,Y 431.18,Z 727.491,A -85,B 0,C 180,E1 19208.262,E2 19208.262} C_VEL
LIN {X 0,Y 430.372,Z 752.963,A -85,B 0,C 180,E1 19207.753,E2 19207.753} C_VEL
LIN {X 0,Y 429.083,Z 773.218,A -85,B 0,C 180,E1 19207.113,E2 19207.113} C_VEL
LIN {X 0,Y 427.269,Z 791.938,A -85,B 0,C 180,E1 19206.303,E2 19206.303} C_VEL
LIN {X 0,Y 424.804,Z 810.897,A -85,B 0,C 180,E1 19205.241,E2 19205.241} C_VEL
LIN {X 0,Y 421.876,Z 829.447,A -85,B 0,C 180,E1 19203.936,E2 19203.936} C_VEL
LIN {X 0,Y 419.178,Z 844.169,A -85,B 0,C 180,E1 19202.687,E2 19202.687} C_VEL
LIN {X 0,Y 417.143,Z 850.638,A -85,B 0,C 180,E1 19202.168,E2 19202.168} C_VEL
LIN {X 0,Y 408.821,Z 866.847,A -85,B 0,C 180,E1 19200.964,E2 19200.964} C_VEL
LIN {X 0,Y 406.647,Z 872.679,A -85,B 0,C 180,E1 19200.333,E2 19200.333} C_VEL
LIN {X 0,Y 402.934,Z 887.213,A -85,B 0,C 180,E1 19198.292,E2 19198.292} C_VEL
LIN {X 0,Y 399.249,Z 901.031,A -85,B 0,C 180,E1 19195.964,E2 19195.964} C_VEL
LIN {X 0,Y 395.921,Z 913.156,A -85,B 0,C 180,E1 19193.517,E2 19193.517} C_VEL
LIN {X 0,Y 392.801,Z 924.531,A -85,B 0,C 180,E1 19190.721,E2 19190.721} C_VEL
LIN {X 0,Y 390.163,Z 934.263,A -85,B 0,C 180,E1 19187.756,E2 19187.756} C_VEL
LIN {X 0,Y 388.228,Z 942.052,A -85,B 0,C 180,E1 19184.772,E2 19184.772} C_VEL
LIN {X 0,Y 386.777,Z 948.431,A -85,B 0,C 180,E1 19181.633,E2 19181.633} C_VEL
LIN {X 0,Y 385.87,Z 953.31,A -85,B 0,C 180,E1 19178.344,E2 19178.344} C_VEL
LIN {X 0,Y 385.383,Z 956.418,A -85,B 0,C 180,E1 19175.21,E2 19175.21} C_VEL
LIN {X 0,Y 385.15,Z 958.122,A -85,B 0,C 180,E1 19171.856,E2 19171.856} C_VEL
LIN {X 0,Y 385.122,Z 958.22,A -85,B 0,C 180,E1 19168.661,E2 19168.661} C_VEL
LIN {X 0,Y 385.304,Z 956.858,A -85,B 0,C 180,E1 19165.386,E2 19165.386} C_VEL
LIN {X 0,Y 385.764,Z 953.947,A -85,B 0,C 180,E1 19162.104,E2 19162.104} C_VEL
LIN {X 0,Y 386.551,Z 949.641,A -85,B 0,C 180,E1 19158.965,E2 19158.965} C_VEL
LIN {X 0,Y 387.925,Z 943.455,A -85,B 0,C 180,E1 19155.726,E2 19155.726} C_VEL
LIN {X 0,Y 389.884,Z 935.406,A -85,B 0,C 180,E1 19152.539,E2 19152.539} C_VEL
LIN {X 0,Y 392.285,Z 926.377,A -85,B 0,C 180,E1 19149.713,E2 19149.713} C_VEL
LIN {X 0,Y 395.097,Z 916.076,A -85,B 0,C 180,E1 19147.063,E2 19147.063} C_VEL
LIN {X 0,Y 398.352,Z 904.449,A -85,B 0,C 180,E1 19144.583,E2 19144.583} C_VEL
LIN {X 0,Y 401.875,Z 891.454,A -85,B 0,C 180,E1 19142.273,E2 19142.273} C_VEL
LIN {X 0,Y 405.599,Z 876.945,A -85,B 0,C 180,E1 19140.135,E2 19140.135} C_VEL
LIN {X 0,Y 409.31,Z 861.413,A -85,B 0,C 180,E1 19138.222,E2 19138.222} C_VEL
LIN {X 0,Y 412.827,Z 845.29,A -85,B 0,C 180,E1 19136.564,E2 19136.564} C_VEL
LIN {X 0,Y 416.242,Z 827.357,A -85,B 0,C 180,E1 19135.047,E2 19135.047} C_VEL
LIN {X 0,Y 419.121,Z 809.26,A -85,B 0,C 180,E1 19133.812,E2 19133.812} C_VEL
LIN {X 0,Y 421.627,Z 789.75,A -85,B 0,C 180,E1 19132.749,E2 19132.749} C_VEL
LIN {X 0,Y 423.514,Z 770.268,A -85,B 0,C 180,E1 19131.935,E2 19131.935} C_VEL
LIN {X 0,Y 424.802,Z 749.524,A -85,B 0,C 180,E1 19131.319,E2 19131.319} C_VEL
LIN {X 0,Y 425.792,Z 713.406,A -85,B 0,C 180,E1 19130.666,E2 19130.666} C_VEL
LIN {X 0,Y 431.597,Z 509.351,A -85,B 0,C 180,E1 19127.205,E2 19127.205} C_VEL
LIN {X 0,Y 426.821,Z 476.764,A -85,B 0,C 180,E1 19125.707,E2 19125.707} C_VEL
LIN {X 0,Y 421.621,Z 468.257,A -85,B 0,C 180,E1 19124.584,E2 19124.584} C_VEL
LIN {X 0,Y 415.123,Z 453.591,A -85,B 0,C 180,E1 19121.665,E2 19121.665} C_VEL
LIN {X 0,Y 409.183,Z 441.38,A -85,B 0,C 180,E1 19118.903,E2 19118.903} C_VEL
LIN {X 0,Y 403.418,Z 429.898,A -85,B 0,C 180,E1 19115.973,E2 19115.973} C_VEL
LIN {X 0,Y 399.98,Z 423.977,A -85,B 0,C 180,E1 19114.226,E2 19114.226} C_VEL
LIN {X 0,Y 397.463,Z 419.46,A -85,B 0,C 180,E1 19112.837,E2 19112.837} C_VEL
LIN {X 0,Y 394.778,Z 414.707,A -85,B 0,C 180,E1 19111.279,E2 19111.279} C_VEL
LIN {X 0,Y 392.558,Z 410.965,A -85,B 0,C 180,E1 19109.949,E2 19109.949} C_VEL
LIN {X 0,Y 391.879,Z 409.687,A -85,B 0,C 180,E1 19109.501,E2 19109.501} C_VEL
LIN {X 0,Y 389.463,Z 406.131,A -85,B 0,C 180,E1 19108.022,E2 19108.022} C_VEL
LIN {X 0,Y 388.704,Z 404.422,A -85,B 0,C 180,E1 19107.416,E2 19107.416} C_VEL
LIN {X 0,Y 386.322,Z 401.535,A -85,B 0,C 180,E1 19105.938,E2 19105.938} C_VEL
LIN {X 0,Y 385.641,Z 399.219,A -85,B 0,C 180,E1 19105,E2 19105} C_VEL
LIN {X 0,Y 385.594,Z 399.004,A -85,B 0,C 180,E1 19101.127,E2 19101.127} C_VEL
LIN {X 0,Y 385.577,Z 399.013,A -85,B 0,C 180,E1 19097.195,E2 19097.195} C_VEL
LIN {X 0,Y 385.565,Z 399.017,A -85,B 0,C 180,E1 19093.344,E2 19093.344} C_VEL
LIN {X 0,Y 385.564,Z 399.021,A -85,B 0,C 180,E1 19089.403,E2 19089.403} C_VEL
LIN {X 0,Y 385.57,Z 399.022,A -85,B 0,C 180,E1 19085.506,E2 19085.506} C_VEL
LIN {X 0,Y 385.588,Z 399.02,A -85,B 0,C 180,E1 19081.635,E2 19081.635} C_VEL
LIN {X 0,Y 385.605,Z 399.017,A -85,B 0,C 180,E1 19077.771,E2 19077.771} C_VEL
LIN {X 0,Y 385.612,Z 399.008,A -85,B 0,C 180,E1 19073.599,E2 19073.599} C_VEL
LIN {X 0,Y 385.597,Z 398.985,A -85,B 0,C 180,E1 19069.543,E2 19069.543} C_VEL
LIN {X 0,Y 385.593,Z 398.952,A -85,B 0,C 180,E1 19065.433,E2 19065.433} C_VEL
LIN {X 0,Y 385.613,Z 399.384,A -85,B 0,C 180,E1 19064.356,E2 19064.356} C_VEL
LIN {X 0,Y 387.373,Z 403.118,A -85,B 0,C 180,E1 19062.888,E2 19062.888} C_VEL
LIN {X 0,Y 389.502,Z 405.304,A -85,B 0,C 180,E1 19061.75,E2 19061.75} C_VEL
LIN {X 0,Y 391.491,Z 409.122,A -85,B 0,C 180,E1 19060.454,E2 19060.454} C_VEL
LIN {X 0,Y 393.192,Z 411.045,A -85,B 0,C 180,E1 19059.612,E2 19059.612} C_VEL
LIN {X 0,Y 395.148,Z 414.715,A -85,B 0,C 180,E1 19058.476,E2 19058.476} C_VEL
LIN {X 0,Y 396.65,Z 416.537,A -85,B 0,C 180,E1 19057.784,E2 19057.784} C_VEL
LIN {X 0,Y 399.127,Z 420.723,A -85,B 0,C 180,E1 19056.528,E2 19056.528} C_VEL
LIN {X 0,Y 400.303,Z 422.602,A -85,B 0,C 180,E1 19055.976,E2 19055.976} C_VEL
LIN {X 0,Y 403.886,Z 428.579,A -85,B 0,C 180,E1 19054.328,E2 19054.328} C_VEL
LIN {X 0,Y 406.393,Z 432.771,A -85,B 0,C 180,E1 19053.242,E2 19053.242} C_VEL
LIN {X 0,Y 411.983,Z 442.282,A -85,B 0,C 180,E1 19050.963,E2 19050.963} C_VEL
LIN {X 0,Y 419.638,Z 456.447,A -85,B 0,C 180,E1 19048.02,E2 19048.02} C_VEL
LIN {X 0,Y 425.335,Z 467.334,A -85,B 0,C 180,E1 19046.062,E2 19046.062} C_VEL
LIN {X 0,Y 436.16,Z 484.268,A -85,B 0,C 180,E1 19043.939,E2 19043.939} C_VEL
LIN {X 0,Y 437.843,Z 507.001,A -85,B 0,C 180,E1 19043.121,E2 19043.121} C_VEL
LIN {X 0,Y 429.799,Z 697.18,A -85,B 0,C 180,E1 19039.393,E2 19039.393} C_VEL
LIN {X 0,Y 425.233,Z 804.65,A -85,B 0,C 180,E1 19037.24,E2 19037.24} C_VEL
LIN {X 0,Y 423.175,Z 828.139,A -85,B 0,C 180,E1 19036.573,E2 19036.573} C_VEL
LIN {X 0,Y 420.537,Z 851.279,A -85,B 0,C 180,E1 19035.697,E2 19035.697} C_VEL
LIN {X 0,Y 417.645,Z 872.66,A -85,B 0,C 180,E1 19034.65,E2 19034.65} C_VEL
LIN {X 0,Y 414.189,Z 895.264,A -85,B 0,C 180,E1 19033.282,E2 19033.282} C_VEL
LIN {X 0,Y 410.609,Z 917.293,A -85,B 0,C 180,E1 19031.665,E2 19031.665} C_VEL
LIN {X 0,Y 407.006,Z 937.58,A -85,B 0,C 180,E1 19029.88,E2 19029.88} C_VEL
LIN {X 0,Y 402.987,Z 959.523,A -85,B 0,C 180,E1 19027.616,E2 19027.616} C_VEL
LIN {X 0,Y 399.511,Z 978.604,A -85,B 0,C 180,E1 19025.319,E2 19025.319} C_VEL
LIN {X 0,Y 396.1,Z 997.231,A -85,B 0,C 180,E1 19022.697,E2 19022.697} C_VEL
LIN {X 0,Y 393.006,Z 1014.9,A -85,B 0,C 180,E1 19019.826,E2 19019.826} C_VEL
LIN {X 0,Y 390.516,Z 1030.404,A -85,B 0,C 180,E1 19016.948,E2 19016.948} C_VEL
LIN {X 0,Y 388.669,Z 1042.575,A -85,B 0,C 180,E1 19014.306,E2 19014.306} C_VEL
LIN {X 0,Y 387.052,Z 1054.388,A -85,B 0,C 180,E1 19011.361,E2 19011.361} C_VEL
LIN {X 0,Y 385.83,Z 1064.589,A -85,B 0,C 180,E1 19008.274,E2 19008.274} C_VEL
LIN {X 0,Y 384.941,Z 1073.453,A -85,B 0,C 180,E1 19005.055,E2 19005.055} C_VEL
LIN {X 0,Y 384.471,Z 1080.05,A -85,B 0,C 180,E1 19002.008,E2 19002.008} C_VEL
LIN {X 0,Y 384.205,Z 1085.421,A -85,B 0,C 180,E1 18998.832,E2 18998.832} C_VEL
LIN {X 0,Y 384.11,Z 1088.981,A -85,B 0,C 180,E1 18995.677,E2 18995.677} C_VEL
LIN {X 0,Y 384.076,Z 1090.835,A -85,B 0,C 180,E1 18992.984,E2 18992.984} C_VEL
LIN {X 0,Y 384.081,Z 1091.598,A -85,B 0,C 180,E1 18989.851,E2 18989.851} C_VEL
LIN {X 0,Y 384.074,Z 1090.759,A -85,B 0,C 180,E1 18986.866,E2 18986.866} C_VEL
LIN {X 0,Y 384.112,Z 1088.851,A -85,B 0,C 180,E1 18984.173,E2 18984.173} C_VEL
LIN {X 0,Y 384.219,Z 1084.953,A -85,B 0,C 180,E1 18980.866,E2 18980.866} C_VEL
LIN {X 0,Y 384.493,Z 1079.766,A -85,B 0,C 180,E1 18977.84,E2 18977.84} C_VEL
LIN {X 0,Y 385.009,Z 1072.708,A -85,B 0,C 180,E1 18974.639,E2 18974.639} C_VEL
LIN {X 0,Y 385.907,Z 1063.885,A -85,B 0,C 180,E1 18971.49,E2 18971.49} C_VEL
LIN {X 0,Y 387.208,Z 1053.22,A -85,B 0,C 180,E1 18968.33,E2 18968.33} C_VEL
LIN {X 0,Y 388.865,Z 1041.273,A -85,B 0,C 180,E1 18965.384,E2 18965.384} C_VEL
LIN {X 0,Y 391.147,Z 1026.389,A -85,B 0,C 180,E1 18962.274,E2 18962.274} C_VEL
LIN {X 0,Y 393.971,Z 1009.508,A -85,B 0,C 180,E1 18959.243,E2 18959.243} C_VEL
LIN {X 0,Y 396.947,Z 992.54,A -85,B 0,C 180,E1 18956.607,E2 18956.607} C_VEL
LIN {X 0,Y 400.391,Z 973.687,A -85,B 0,C 180,E1 18954.066,E2 18954.066} C_VEL
LIN {X 0,Y 404.009,Z 954.076,A -85,B 0,C 180,E1 18951.778,E2 18951.778} C_VEL
LIN {X 0,Y 407.733,Z 933.481,A -85,B 0,C 180,E1 18949.737,E2 18949.737} C_VEL
LIN {X 0,Y 411.532,Z 911.502,A -85,B 0,C 180,E1 18947.888,E2 18947.888} C_VEL
LIN {X 0,Y 415.088,Z 889.861,A -85,B 0,C 180,E1 18946.36,E2 18946.36} C_VEL
LIN {X 0,Y 418.198,Z 868.717,A -85,B 0,C 180,E1 18945.145,E2 18945.145} C_VEL
LIN {X 0,Y 421.222,Z 845.502,A -85,B 0,C 180,E1 18944.062,E2 18944.062} C_VEL
LIN {X 0,Y 423.597,Z 823.833,A -85,B 0,C 180,E1 18943.29,E2 18943.29} C_VEL
LIN {X 0,Y 425.495,Z 799.351,A -85,B 0,C 180,E1 18942.646,E2 18942.646} C_VEL
LIN {X 0,Y 433.988,Z 597.651,A -85,B 0,C 180,E1 18938.649,E2 18938.649} C_VEL
LIN {X 0,Y 437.745,Z 504.283,A -85,B 0,C 180,E1 18936.808,E2 18936.808} C_VEL
LIN {X 0,Y 435.963,Z 483.906,A -85,B 0,C 180,E1 18936.034,E2 18936.034} C_VEL
LIN {X 0,Y 424.571,Z 466.073,A -85,B 0,C 180,E1 18933.764,E2 18933.764} C_VEL
LIN {X 0,Y 416.184,Z 449.872,A -85,B 0,C 180,E1 18930.698,E2 18930.698} C_VEL
LIN {X 0,Y 410.181,Z 439.308,A -85,B 0,C 180,E1 18928.36,E2 18928.36} C_VEL
LIN {X 0,Y 404.759,Z 430.004,A -85,B 0,C 180,E1 18926.085,E2 18926.085} C_VEL
LIN {X 0,Y 401.973,Z 425.432,A -85,B 0,C 180,E1 18924.857,E2 18924.857} C_VEL
LIN {X 0,Y 399.293,Z 420.911,A -85,B 0,C 180,E1 18923.58,E2 18923.58} C_VEL
LIN {X 0,Y 396.753,Z 416.904,A -85,B 0,C 180,E1 18922.349,E2 18922.349} C_VEL
LIN {X 0,Y 395.969,Z 415.632,A -85,B 0,C 180,E1 18921.944,E2 18921.944} C_VEL
LIN {X 0,Y 393.519,Z 411.98,A -85,B 0,C 180,E1 18920.681,E2 18920.681} C_VEL
LIN {X 0,Y 392.87,Z 410.457,A -85,B 0,C 180,E1 18920.25,E2 18920.25} C_VEL
LIN {X 0,Y 390.388,Z 407.522,A -85,B 0,C 180,E1 18918.981,E2 18918.981} C_VEL
LIN {X 0,Y 389.179,Z 404.792,A -85,B 0,C 180,E1 18918.111,E2 18918.111} C_VEL
LIN {X 0,Y 386.385,Z 401.631,A -85,B 0,C 180,E1 18916.537,E2 18916.537} C_VEL
LIN {X 0,Y 385.597,Z 399.304,A -85,B 0,C 180,E1 18915.644,E2 18915.644} C_VEL
LIN {X 0,Y 385.567,Z 398.937,A -85,B 0,C 180,E1 18913.038,E2 18913.038} C_VEL
LIN {X 0,Y 385.563,Z 399.01,A -85,B 0,C 180,E1 18909.101,E2 18909.101} C_VEL
LIN {X 0,Y 385.554,Z 399.008,A -85,B 0,C 180,E1 18905.207,E2 18905.207} C_VEL
LIN {X 0,Y 385.553,Z 399.007,A -85,B 0,C 180,E1 18901.188,E2 18901.188} C_VEL
LIN {X 0,Y 385.558,Z 399.005,A -85,B 0,C 180,E1 18897.175,E2 18897.175} C_VEL
LIN {X 0,Y 385.571,Z 399.002,A -85,B 0,C 180,E1 18893.298,E2 18893.298} C_VEL
LIN {X 0,Y 385.593,Z 398.999,A -85,B 0,C 180,E1 18889.391,E2 18889.391} C_VEL
LIN {X 0,Y 385.618,Z 398.995,A -85,B 0,C 180,E1 18885.433,E2 18885.433} C_VEL
LIN {X 0,Y 385.602,Z 398.997,A -85,B 0,C 180,E1 18881.401,E2 18881.401} C_VEL
LIN {X 0,Y 385.587,Z 399.001,A -85,B 0,C 180,E1 18877.432,E2 18877.432} C_VEL
LIN {X 0,Y 385.633,Z 399.239,A -85,B 0,C 180,E1 18874.808,E2 18874.808} C_VEL
LIN {X 0,Y 387.176,Z 402.89,A -85,B 0,C 180,E1 18873.298,E2 18873.298} C_VEL
LIN {X 0,Y 389.167,Z 405.241,A -85,B 0,C 180,E1 18872.107,E2 18872.107} C_VEL
LIN {X 0,Y 391.087,Z 408.847,A -85,B 0,C 180,E1 18870.77,E2 18870.77} C_VEL
LIN {X 0,Y 392.42,Z 410.552,A -85,B 0,C 180,E1 18870.032,E2 18870.032} C_VEL
LIN {X 0,Y 394.829,Z 414.787,A -85,B 0,C 180,E1 18868.555,E2 18868.555} C_VEL
LIN {X 0,Y 398.608,Z 421.505,A -85,B 0,C 180,E1 18866.386,E2 18866.386} C_VEL
LIN {X 0,Y 401.416,Z 426.609,A -85,B 0,C 180,E1 18864.873,E2 18864.873} C_VEL
LIN {X 0,Y 406.033,Z 435.094,A -85,B 0,C 180,E1 18862.537,E2 18862.537} C_VEL
LIN {X 0,Y 412.081,Z 447.215,A -85,B 0,C 180,E1 18859.621,E2 18859.621} C_VEL
LIN {X 0,Y 418.468,Z 461.015,A -85,B 0,C 180,E1 18856.706,E2 18856.706} C_VEL
LIN {X 0,Y 422.292,Z 469.694,A -85,B 0,C 180,E1 18855.097,E2 18855.097} C_VEL
LIN {X 0,Y 426.997,Z 477.353,A -85,B 0,C 180,E1 18854.147,E2 18854.147} C_VEL
LIN {X 0,Y 431.561,Z 510.526,A -85,B 0,C 180,E1 18852.671,E2 18852.671} C_VEL
LIN {X 0,Y 425.262,Z 733.214,A -85,B 0,C 180,E1 18848.91,E2 18848.91} C_VEL
LIN {X 0,Y 424.452,Z 755.162,A -85,B 0,C 180,E1 18848.439,E2 18848.439} C_VEL
LIN {X 0,Y 422.953,Z 776.328,A -85,B 0,C 180,E1 18847.738,E2 18847.738} C_VEL
LIN {X 0,Y 421.08,Z 794.564,A -85,B 0,C 180,E1 18846.924,E2 18846.924} C_VEL
LIN {X 0,Y 418.457,Z 813.457,A -85,B 0,C 180,E1 18845.832,E2 18845.832} C_VEL
LIN {X 0,Y 415.439,Z 831.507,A -85,B 0,C 180,E1 18844.527,E2 18844.527} C_VEL
LIN {X 0,Y 412.073,Z 848.759,A -85,B 0,C 180,E1 18843.007,E2 18843.007} C_VEL
LIN {X 0,Y 408.451,Z 865.148,A -85,B 0,C 180,E1 18841.263,E2 18841.263} C_VEL
LIN {X 0,Y 406.647,Z 872.679,A -85,B 0,C 180,E1 18840.333,E2 18840.333} C_VEL
LIN {X 0,Y 404.445,Z 878.467,A -85,B 0,C 180,E1 18839.67,E2 18839.67} C_VEL
LIN {X 0,Y 395.718,Z 892.913,A -85,B 0,C 180,E1 18838.085,E2 18838.085} C_VEL
LIN {X 0,Y 393.493,Z 897.983,A -85,B 0,C 180,E1 18837.31,E2 18837.31} C_VEL
LIN {X 0,Y 389.885,Z 910.545,A -85,B 0,C 180,E1 18834.871,E2 18834.871} C_VEL
LIN {X 0,Y 386.492,Z 922.149,A -85,B 0,C 180,E1 18832.157,E2 18832.157} C_VEL
LIN {X 0,Y 383.668,Z 932.059,A -85,B 0,C 180,E1 18829.328,E2 18829.328} C_VEL
LIN {X 0,Y 381.325,Z 940.622,A -85,B 0,C 180,E1 18826.294,E2 18826.294} C_VEL
LIN {X 0,Y 379.551,Z 947.638,A -85,B 0,C 180,E1 18823.094,E2 18823.094} C_VEL
LIN {X 0,Y 378.388,Z 952.915,A -85,B 0,C 180,E1 18819.89,E2 18819.89} C_VEL
LIN {X 0,Y 377.685,Z 956.757,A -85,B 0,C 180,E1 18816.537,E2 18816.537} C_VEL
LIN {X 0,Y 377.323,Z 959.003,A -85,B 0,C 180,E1 18813.19,E2 18813.19} C_VEL
LIN {X 0,Y 377.236,Z 959.738,A -85,B 0,C 180,E1 18809.848,E2 18809.848} C_VEL
LIN {X 0,Y 377.341,Z 958.928,A -85,B 0,C 180,E1 18806.506,E2 18806.506} C_VEL
LIN {X 0,Y 377.725,Z 956.574,A -85,B 0,C 180,E1 18803.159,E2 18803.159} C_VEL
LIN {X 0,Y 378.445,Z 952.619,A -85,B 0,C 180,E1 18799.804,E2 18799.804} C_VEL
LIN {X 0,Y 379.721,Z 946.912,A -85,B 0,C 180,E1 18796.447,E2 18796.447} C_VEL
LIN {X 0,Y 381.462,Z 940.065,A -85,B 0,C 180,E1 18793.399,E2 18793.399} C_VEL
LIN {X 0,Y 383.873,Z 931.419,A -85,B 0,C 180,E1 18790.366,E2 18790.366} C_VEL
LIN {X 0,Y 386.783,Z 921.231,A -85,B 0,C 180,E1 18787.506,E2 18787.506} C_VEL
LIN {X 0,Y 389.986,Z 910.27,A -85,B 0,C 180,E1 18784.974,E2 18784.974} C_VEL
LIN {X 0,Y 393.706,Z 897.27,A -85,B 0,C 180,E1 18782.47,E2 18782.47} C_VEL
LIN {X 0,Y 397.634,Z 883.206,A -85,B 0,C 180,E1 18780.223,E2 18780.223} C_VEL
LIN {X 0,Y 401.637,Z 867.522,A -85,B 0,C 180,E1 18778.145,E2 18778.145} C_VEL
LIN {X 0,Y 405.403,Z 851.367,A -85,B 0,C 180,E1 18776.379,E2 18776.379} C_VEL
LIN {X 0,Y 409.071,Z 833.602,A -85,B 0,C 180,E1 18774.771,E2 18774.771} C_VEL
LIN {X 0,Y 412.217,Z 815.836,A -85,B 0,C 180,E1 18773.453,E2 18773.453} C_VEL
LIN {X 0,Y 414.929,Z 797.16,A -85,B 0,C 180,E1 18772.348,E2 18772.348} C_VEL
LIN {X 0,Y 417.074,Z 777.813,A -85,B 0,C 180,E1 18771.458,E2 18771.458} C_VEL
LIN {X 0,Y 418.652,Z 757.015,A -85,B 0,C 180,E1 18770.752,E2 18770.752} C_VEL
LIN {X 0,Y 419.514,Z 736.104,A -85,B 0,C 180,E1 18770.282,E2 18770.282} C_VEL
LIN {X 0,Y 426.245,Z 512.491,A -85,B 0,C 180,E1 18766.461,E2 18766.461} C_VEL
LIN {X 0,Y 425.714,Z 506.98,A -85,B 0,C 180,E1 18766.25,E2 18766.25} C_VEL
LIN {X 0,Y 422.012,Z 481.208,A -85,B 0,C 180,E1 18765.034,E2 18765.034} C_VEL
LIN {X 0,Y 413.998,Z 468.652,A -85,B 0,C 180,E1 18763.307,E2 18763.307} C_VEL
LIN {X 0,Y 408.2,Z 455.693,A -85,B 0,C 180,E1 18760.595,E2 18760.595} C_VEL
LIN {X 0,Y 402.279,Z 443.469,A -85,B 0,C 180,E1 18757.693,E2 18757.693} C_VEL
LIN {X 0,Y 397.408,Z 434.284,A -85,B 0,C 180,E1 18755.181,E2 18755.181} C_VEL
LIN {X 0,Y 395.06,Z 429.919,A -85,B 0,C 180,E1 18753.887,E2 18753.887} C_VEL
LIN {X 0,Y 392.78,Z 425.735,A -85,B 0,C 180,E1 18752.585,E2 18752.585} C_VEL
LIN {X 0,Y 390.149,Z 421.023,A -85,B 0,C 180,E1 18751.006,E2 18751.006} C_VEL
LIN {X 0,Y 387.826,Z 416.698,A -85,B 0,C 180,E1 18749.5,E2 18749.5} C_VEL
LIN {X 0,Y 385.158,Z 412.848,A -85,B 0,C 180,E1 18747.858,E2 18747.858} C_VEL
LIN {X 0,Y 384.204,Z 410.914,A -85,B 0,C 180,E1 18747.123,E2 18747.123} C_VEL
LIN {X 0,Y 381.91,Z 407.824,A -85,B 0,C 180,E1 18745.594,E2 18745.594} C_VEL
LIN {X 0,Y 380.91,Z 405.513,A -85,B 0,C 180,E1 18744.669,E2 18744.669} C_VEL
LIN {X 0,Y 378.587,Z 402.828,A -85,B 0,C 180,E1 18743.009,E2 18743.009} C_VEL
LIN {X 0,Y 377.666,Z 400.281,A -85,B 0,C 180,E1 18741.756,E2 18741.756} C_VEL
LIN {X 0,Y 377.663,Z 399.985,A -85,B 0,C 180,E1 18738.524,E2 18738.524} C_VEL
LIN {X 0,Y 377.679,Z 399.983,A -85,B 0,C 180,E1 18734.567,E2 18734.567} C_VEL
LIN {X 0,Y 377.666,Z 399.987,A -85,B 0,C 180,E1 18730.372,E2 18730.372} C_VEL
LIN {X 0,Y 377.673,Z 399.991,A -85,B 0,C 180,E1 18726.232,E2 18726.232} C_VEL
LIN {X 0,Y 377.662,Z 399.997,A -85,B 0,C 180,E1 18722.125,E2 18722.125} C_VEL
LIN {X 0,Y 377.645,Z 400.003,A -85,B 0,C 180,E1 18718.18,E2 18718.18} C_VEL
LIN {X 0,Y 377.632,Z 400.009,A -85,B 0,C 180,E1 18714.226,E2 18714.226} C_VEL
LIN {X 0,Y 377.622,Z 400.004,A -85,B 0,C 180,E1 18710.244,E2 18710.244} C_VEL
LIN {X 0,Y 377.694,Z 400.308,A -85,B 0,C 180,E1 18707.696,E2 18707.696} C_VEL
LIN {X 0,Y 379.475,Z 404.139,A -85,B 0,C 180,E1 18705.843,E2 18705.843} C_VEL
LIN {X 0,Y 381.608,Z 406.308,A -85,B 0,C 180,E1 18704.5,E2 18704.5} C_VEL
LIN {X 0,Y 383.561,Z 410.093,A -85,B 0,C 180,E1 18703.025,E2 18703.025} C_VEL
LIN {X 0,Y 385.412,Z 411.979,A -85,B 0,C 180,E1 18702.019,E2 18702.019} C_VEL
LIN {X 0,Y 387.382,Z 415.789,A -85,B 0,C 180,E1 18700.709,E2 18700.709} C_VEL
LIN {X 0,Y 389.044,Z 417.772,A -85,B 0,C 180,E1 18699.856,E2 18699.856} C_VEL
LIN {X 0,Y 391.306,Z 421.737,A -85,B 0,C 180,E1 18698.569,E2 18698.569} C_VEL
LIN {X 0,Y 392.471,Z 423.292,A -85,B 0,C 180,E1 18698.007,E2 18698.007} C_VEL
LIN {X 0,Y 395.275,Z 427.751,A -85,B 0,C 180,E1 18696.601,E2 18696.601} C_VEL
LIN {X 0,Y 401.489,Z 438.276,A -85,B 0,C 180,E1 18693.707,E2 18693.707} C_VEL
LIN {X 0,Y 408.633,Z 450.833,A -85,B 0,C 180,E1 18690.702,E2 18690.702} C_VEL
LIN {X 0,Y 416.934,Z 466.606,A -85,B 0,C 180,E1 18687.509,E2 18687.509} C_VEL
LIN {X 0,Y 428.943,Z 485.091,A -85,B 0,C 180,E1 18685.011,E2 18685.011} C_VEL
LIN {X 0,Y 431.055,Z 488.821,A -85,B 0,C 180,E1 18684.588,E2 18684.588} C_VEL
LIN {X 0,Y 432.406,Z 508.304,A -85,B 0,C 180,E1 18683.88,E2 18683.88} C_VEL
LIN {X 0,Y 424.021,Z 697.992,A -85,B 0,C 180,E1 18680.129,E2 18680.129} C_VEL
LIN {X 0,Y 419.313,Z 803.897,A -85,B 0,C 180,E1 18677.985,E2 18677.985} C_VEL
LIN {X 0,Y 417.18,Z 827.405,A -85,B 0,C 180,E1 18677.312,E2 18677.312} C_VEL
LIN {X 0,Y 414.425,Z 850.493,A -85,B 0,C 180,E1 18676.431,E2 18676.431} C_VEL
LIN {X 0,Y 411.445,Z 871.607,A -85,B 0,C 180,E1 18675.389,E2 18675.389} C_VEL
LIN {X 0,Y 407.673,Z 895.018,A -85,B 0,C 180,E1 18673.955,E2 18673.955} C_VEL
LIN {X 0,Y 403.917,Z 916.858,A -85,B 0,C 180,E1 18672.323,E2 18672.323} C_VEL
LIN {X 0,Y 400.144,Z 937.044,A -85,B 0,C 180,E1 18670.517,E2 18670.517} C_VEL
